KUKA KRL program: EPS_2_25716_MHDA01_A_20260123031854.src

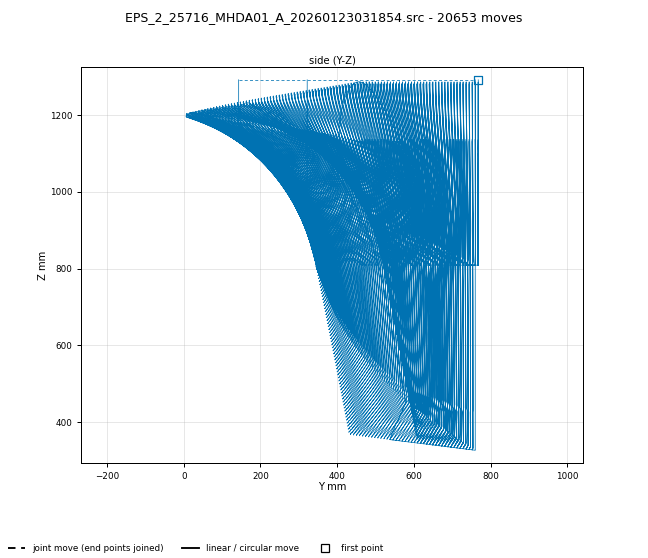
[picture p0: tool path of EPS_2_25716_MHDA01_A_20260123031854.src, 20653 of 20655 moves have a stored position in this frame; points joined in program order, loops and branches not executed]
&ACCESS RVP
&REL 4
&COMMENT QRS 19112012
&PARAM EDITMASK = *
DEF PART()
EXT BAS (BAS_COMMAND :IN,REAL :IN )
INT I
BAS (#INITMOV,0 )

;KUKA QRS Post kuka4.cps  Date:22-06-2017 !

File_ID=3001

QRS_PRE_INIT()

;Init var - Until changes are made in qrs_pre_init
Outlet_Square_prg=0
Inlet_1_Square_prg=0
Inlet_2_Square_prg=0
Inlet_3_Square_prg=0
Inlet_4_Square_prg=0
Inlet_5_Square_prg=0

Outlet_1={X 0.000, Y 457.000, Z 863.000, B 0.000, E1 0.000 }
Inlet_1={X 0.000, Y 457.000, Z 713.000, B 0.000, E1 245.000 }
Outlet_1_type=838
Inlet_1_type=838
;QRS#1=Sidecore dimensions
;QRS#2=825-33" Concrete
;QRS#3=825-33" Concrete
;QRS#4=
;QRS#5=
;QRS#6=
;QRS#7=
;QRS#8=
;QRS#9=S306-46
;QRS#10=S306-46
;QRS#11=
;QRS#12=
;QRS#13=
;QRS#14=
;QRS#15=
;QRS#16=1524x152x1753 5,75'
;QRS#17=EPS Height
;QRS#18=1282
;QRS#19=*
;QRS#20= UPDATED VERSION 22-06-2017
;QRS#21=*
Outlet_Square=0650
Inlet_1_Square=0650
Inlet_2_Square=0
Inlet_3_Square=0
Inlet_4_Square=0
Inlet_5_Square=0
Mill_Square=1
Outlet_Square_Prg=267
Inlet_1_Square_prg=267

QRS_INIT()

$ADVANCE=5

; T1
PTP {E1 173.029,E2 173.029}
PTP {X 0,Y 767.722,A -85,B 0,C 180,E1 173.029,E2 173.029,E3 0,E4 0,E5 0,E6 0}
QRS_SPEED_INIT()
LIN {X 0,Y 767.722,Z 1292,A -85,B 0,C 180,E1 173.029,E2 173.029,E3 0,E4 0,E5 0,E6 0} C_VEL
LIN {X 0,Y 767.722,Z 811.06,A -85,B 0,C 180,E1 173.029,E2 173.029} C_VEL
LIN {X 0,Y 767.749,Z 809.06,A -85,B 0,C 180,E1 173.179,E2 173.179} C_VEL
LIN {X 0,Y 767.812,Z 809.06,A -85,B 0,C 180,E1 173.458,E2 173.458} C_VEL
LIN {X 0,Y 767.844,Z 809.06,A -85,B 0,C 180,E1 177.201,E2 177.201} C_VEL
LIN {X 0,Y 767.885,Z 809.06,A -85,B 0,C 180,E1 180.933,E2 180.933} C_VEL
LIN {X 0,Y 767.853,Z 809.06,A -85,B 0,C 180,E1 184.668,E2 184.668} C_VEL
LIN {X 0,Y 767.842,Z 809.06,A -85,B 0,C 180,E1 188.423,E2 188.423} C_VEL
LIN {X 0,Y 767.815,Z 809.06,A -85,B 0,C 180,E1 192.216,E2 192.216} C_VEL
LIN {X 0,Y 767.835,Z 809.06,A -85,B 0,C 180,E1 196.207,E2 196.207} C_VEL
LIN {X 0,Y 767.767,Z 809.06,A -85,B 0,C 180,E1 199.988,E2 199.988} C_VEL
LIN {X 0,Y 767.76,Z 809.06,A -85,B 0,C 180,E1 204.012,E2 204.012} C_VEL
LIN {X 0,Y 767.747,Z 809.06,A -85,B 0,C 180,E1 208.167,E2 208.167} C_VEL
LIN {X 0,Y 767.299,Z 809.06,A -85,B 0,C 180,E1 210.325,E2 210.325} C_VEL
LIN {X 0,Y 767.722,Z 809.06,A -85,B 0,C 180,E1 212.492,E2 212.492} C_VEL
LIN {X 0,Y 767.413,Z 809.06,A -85,B 0,C 180,E1 213.849,E2 213.849} C_VEL
LIN {X 0,Y 767.746,Z 809.06,A -85,B 0,C 180,E1 217.099,E2 217.099} C_VEL
LIN {X 0,Y 767.186,Z 809.06,A -85,B 0,C 180,E1 220.04,E2 220.04} C_VEL
LIN {X 0,Y 767.672,Z 809.06,A -85,B 0,C 180,E1 221.87,E2 221.87} C_VEL
LIN {X 0,Y 767.699,Z 809.06,A -85,B 0,C 180,E1 222.901,E2 222.901} C_VEL
LIN {X 0,Y 767.698,Z 809.06,A -85,B 0,C 180,E1 224.426,E2 224.426} C_VEL
LIN {X 0,Y 767.66,Z 809.06,A -85,B 0,C 180,E1 225.572,E2 225.572} C_VEL
LIN {X 0,Y 767.698,Z 809.06,A -85,B 0,C 180,E1 229.916,E2 229.916} C_VEL
LIN {X 0,Y 767.769,Z 809.06,A -85,B 0,C 180,E1 230.595,E2 230.595} C_VEL
LIN {X 0,Y 767.848,Z 809.06,A -85,B 0,C 180,E1 233.269,E2 233.269} C_VEL
LIN {X 0,Y 766.331,Z 809.06,A -85,B 0,C 180,E1 233.48,E2 233.48} C_VEL
LIN {X 0,Y 767.104,Z 827.55,A -85,B 0,C 180,E1 233.745,E2 233.745} C_VEL
LIN {X 0,Y 767.17,Z 886.209,A -85,B 0,C 180,E1 234.412,E2 234.412} C_VEL
LIN {X 0,Y 767.458,Z 906.942,A -85,B 0,C 180,E1 234.685,E2 234.685} C_VEL
LIN {X 0,Y 767.407,Z 923.144,A -85,B 0,C 180,E1 234.938,E2 234.938} C_VEL
LIN {X 0,Y 767.212,Z 935.539,A -85,B 0,C 180,E1 235.164,E2 235.164} C_VEL
LIN {X 0,Y 767.339,Z 953.521,A -85,B 0,C 180,E1 235.567,E2 235.567} C_VEL
LIN {X 0,Y 767.292,Z 964.717,A -85,B 0,C 180,E1 235.849,E2 235.849} C_VEL
LIN {X 0,Y 767.46,Z 977.757,A -85,B 0,C 180,E1 236.229,E2 236.229} C_VEL
LIN {X 0,Y 767.482,Z 994.943,A -85,B 0,C 180,E1 236.765,E2 236.765} C_VEL
LIN {X 0,Y 767.407,Z 1008.2,A -85,B 0,C 180,E1 237.226,E2 237.226} C_VEL
LIN {X 0,Y 767.51,Z 1017.146,A -85,B 0,C 180,E1 237.568,E2 237.568} C_VEL
LIN {X 0,Y 767.581,Z 1032.615,A -85,B 0,C 180,E1 238.19,E2 238.19} C_VEL
LIN {X 0,Y 767.446,Z 1051.001,A -85,B 0,C 180,E1 239.004,E2 239.004} C_VEL
LIN {X 0,Y 767.587,Z 1068.192,A -85,B 0,C 180,E1 239.855,E2 239.855} C_VEL
LIN {X 0,Y 767.618,Z 1085.156,A -85,B 0,C 180,E1 240.771,E2 240.771} C_VEL
LIN {X 0,Y 767.607,Z 1101.948,A -85,B 0,C 180,E1 241.761,E2 241.761} C_VEL
LIN {X 0,Y 767.626,Z 1117.369,A -85,B 0,C 180,E1 242.75,E2 242.75} C_VEL
LIN {X 0,Y 767.651,Z 1132.728,A -85,B 0,C 180,E1 243.819,E2 243.819} C_VEL
LIN {X 0,Y 767.584,Z 1147.859,A -85,B 0,C 180,E1 244.959,E2 244.959} C_VEL
LIN {X 0,Y 767.612,Z 1160.458,A -85,B 0,C 180,E1 245.983,E2 245.983} C_VEL
LIN {X 0,Y 767.704,Z 1173.515,A -85,B 0,C 180,E1 247.13,E2 247.13} C_VEL
LIN {X 0,Y 767.583,Z 1186.75,A -85,B 0,C 180,E1 248.384,E2 248.384} C_VEL
LIN {X 0,Y 767.736,Z 1199.104,A -85,B 0,C 180,E1 249.665,E2 249.665} C_VEL
LIN {X 0,Y 767.55,Z 1210.953,A -85,B 0,C 180,E1 250.996,E2 250.996} C_VEL
LIN {X 0,Y 767.566,Z 1220.98,A -85,B 0,C 180,E1 252.225,E2 252.225} C_VEL
LIN {X 0,Y 767.803,Z 1230.047,A -85,B 0,C 180,E1 253.451,E2 253.451} C_VEL
LIN {X 0,Y 767.523,Z 1241.12,A -85,B 0,C 180,E1 255.092,E2 255.092} C_VEL
LIN {X 0,Y 767.763,Z 1249.724,A -85,B 0,C 180,E1 256.547,E2 256.547} C_VEL
LIN {X 0,Y 767.583,Z 1255.072,A -85,B 0,C 180,E1 257.542,E2 257.542} C_VEL
LIN {X 0,Y 767.466,Z 1258.642,A -85,B 0,C 180,E1 258.256,E2 258.256} C_VEL
LIN {X 0,Y 767.574,Z 1264.125,A -85,B 0,C 180,E1 259.446,E2 259.446} C_VEL
LIN {X 0,Y 767.772,Z 1266.941,A -85,B 0,C 180,E1 260.159,E2 260.159} C_VEL
LIN {X 0,Y 767.609,Z 1270.613,A -85,B 0,C 180,E1 261.103,E2 261.103} C_VEL
LIN {X 0,Y 767.526,Z 1275.33,A -85,B 0,C 180,E1 262.515,E2 262.515} C_VEL
LIN {X 0,Y 767.729,Z 1277.921,A -85,B 0,C 180,E1 263.457,E2 263.457} C_VEL
LIN {X 0,Y 767.753,Z 1279.763,A -85,B 0,C 180,E1 264.208,E2 264.208} C_VEL
LIN {X 0,Y 767.526,Z 1282.157,A -85,B 0,C 180,E1 265.33,E2 265.33} C_VEL
LIN {X 0,Y 767.596,Z 1283.961,A -85,B 0,C 180,E1 266.453,E2 266.453} C_VEL
LIN {X 0,Y 767.784,Z 1284.832,A -85,B 0,C 180,E1 267.201,E2 267.201} C_VEL
LIN {X 0,Y 767.485,Z 1286.213,A -85,B 0,C 180,E1 269.067,E2 269.067} C_VEL
LIN {X 0,Y 767.799,Z 1286.153,A -85,B 0,C 180,E1 270.932,E2 270.932} C_VEL
LIN {X 0,Y 767.787,Z 1284.832,A -85,B 0,C 180,E1 272.799,E2 272.799} C_VEL
LIN {X 0,Y 767.6,Z 1283.418,A -85,B 0,C 180,E1 273.921,E2 273.921} C_VEL
LIN {X 0,Y 767.502,Z 1282.163,A -85,B 0,C 180,E1 274.67,E2 274.67} C_VEL
LIN {X 0,Y 767.612,Z 1279.789,A -85,B 0,C 180,E1 275.793,E2 275.793} C_VEL
LIN {X 0,Y 767.819,Z 1277.906,A -85,B 0,C 180,E1 276.542,E2 276.542} C_VEL
LIN {X 0,Y 767.57,Z 1275.324,A -85,B 0,C 180,E1 277.484,E2 277.484} C_VEL
LIN {X 0,Y 767.464,Z 1270.637,A -85,B 0,C 180,E1 278.899,E2 278.899} C_VEL
LIN {X 0,Y 767.675,Z 1266.958,A -85,B 0,C 180,E1 279.842,E2 279.842} C_VEL
LIN {X 0,Y 767.812,Z 1264.091,A -85,B 0,C 180,E1 280.55,E2 280.55} C_VEL
LIN {X 0,Y 767.541,Z 1256.36,A -85,B 0,C 180,E1 282.22,E2 282.22} C_VEL
LIN {X 0,Y 767.797,Z 1247.861,A -85,B 0,C 180,E1 283.778,E2 283.778} C_VEL
LIN {X 0,Y 767.526,Z 1239.921,A -85,B 0,C 180,E1 285.1,E2 285.1} C_VEL
LIN {X 0,Y 767.65,Z 1230.061,A -85,B 0,C 180,E1 286.552,E2 286.552} C_VEL
LIN {X 0,Y 767.763,Z 1224.604,A -85,B 0,C 180,E1 287.281,E2 287.281} C_VEL
LIN {X 0,Y 767.618,Z 1219.008,A -85,B 0,C 180,E1 288.018,E2 288.018} C_VEL
LIN {X 0,Y 767.578,Z 1208.865,A -85,B 0,C 180,E1 289.25,E2 289.25} C_VEL
LIN {X 0,Y 767.782,Z 1196.924,A -85,B 0,C 180,E1 290.566,E2 290.566} C_VEL
LIN {X 0,Y 767.586,Z 1184.113,A -85,B 0,C 180,E1 291.872,E2 291.872} C_VEL
LIN {X 0,Y 767.66,Z 1172.11,A -85,B 0,C 180,E1 292.998,E2 292.998} C_VEL
LIN {X 0,Y 767.691,Z 1158.934,A -85,B 0,C 180,E1 294.142,E2 294.142} C_VEL
LIN {X 0,Y 767.62,Z 1144.01,A -85,B 0,C 180,E1 295.338,E2 295.338} C_VEL
LIN {X 0,Y 767.652,Z 1129.639,A -85,B 0,C 180,E1 296.401,E2 296.401} C_VEL
LIN {X 0,Y 767.615,Z 1114.367,A -85,B 0,C 180,E1 297.447,E2 297.447} C_VEL
LIN {X 0,Y 767.599,Z 1098.637,A -85,B 0,C 180,E1 298.44,E2 298.44} C_VEL
LIN {X 0,Y 767.566,Z 1083.423,A -85,B 0,C 180,E1 299.33,E2 299.33} C_VEL
LIN {X 0,Y 767.575,Z 1064.92,A -85,B 0,C 180,E1 300.312,E2 300.312} C_VEL
LIN {X 0,Y 767.441,Z 1046.6,A -85,B 0,C 180,E1 301.2,E2 301.2} C_VEL
LIN {X 0,Y 767.574,Z 1029.388,A -85,B 0,C 180,E1 301.947,E2 301.947} C_VEL
LIN {X 0,Y 767.522,Z 1009.76,A -85,B 0,C 180,E1 302.714,E2 302.714} C_VEL
LIN {X 0,Y 767.358,Z 997.436,A -85,B 0,C 180,E1 303.153,E2 303.153} C_VEL
LIN {X 0,Y 767.471,Z 988.18,A -85,B 0,C 180,E1 303.452,E2 303.452} C_VEL
LIN {X 0,Y 767.491,Z 969.899,A -85,B 0,C 180,E1 303.999,E2 303.999} C_VEL
LIN {X 0,Y 767.246,Z 953.494,A -85,B 0,C 180,E1 304.438,E2 304.438} C_VEL
LIN {X 0,Y 767.411,Z 935.529,A -85,B 0,C 180,E1 304.826,E2 304.826} C_VEL
LIN {X 0,Y 767.255,Z 918.227,A -85,B 0,C 180,E1 305.152,E2 305.152} C_VEL
LIN {X 0,Y 767.195,Z 912.098,A -85,B 0,C 180,E1 305.255,E2 305.255} C_VEL
LIN {X 0,Y 767.34,Z 895.861,A -85,B 0,C 180,E1 305.467,E2 305.467} C_VEL
LIN {X 0,Y 767.184,Z 847.286,A -85,B 0,C 180,E1 306.027,E2 306.027} C_VEL
LIN {X 0,Y 766.354,Z 809.06,A -85,B 0,C 180,E1 306.518,E2 306.518} C_VEL
LIN {X 0,Y 767.867,Z 809.06,A -85,B 0,C 180,E1 307.025,E2 307.025} C_VEL
LIN {X 0,Y 767.157,Z 809.06,A -85,B 0,C 180,E1 310.036,E2 310.036} C_VEL
LIN {X 0,Y 767.638,Z 809.06,A -85,B 0,C 180,E1 311.871,E2 311.871} C_VEL
LIN {X 0,Y 767.679,Z 809.06,A -85,B 0,C 180,E1 312.899,E2 312.899} C_VEL
LIN {X 0,Y 767.687,Z 809.06,A -85,B 0,C 180,E1 314.425,E2 314.425} C_VEL
LIN {X 0,Y 767.662,Z 809.06,A -85,B 0,C 180,E1 315.572,E2 315.572} C_VEL
LIN {X 0,Y 767.695,Z 809.06,A -85,B 0,C 180,E1 319.914,E2 319.914} C_VEL
LIN {X 0,Y 767.699,Z 809.06,A -85,B 0,C 180,E1 320.59,E2 320.59} C_VEL
LIN {X 0,Y 767.222,Z 809.06,A -85,B 0,C 180,E1 322.952,E2 322.952} C_VEL
LIN {X 0,Y 767.706,Z 809.06,A -85,B 0,C 180,E1 325.267,E2 325.267} C_VEL
LIN {X 0,Y 767.75,Z 809.06,A -85,B 0,C 180,E1 329.62,E2 329.62} C_VEL
LIN {X 0,Y 767.63,Z 809.06,A -85,B 0,C 180,E1 333.924,E2 333.924} C_VEL
LIN {X 0,Y 767.153,Z 809.06,A -85,B 0,C 180,E1 335.967,E2 335.967} C_VEL
LIN {X 0,Y 767.108,Z 809.06,A -85,B 0,C 180,E1 338.214,E2 338.214} C_VEL
LIN {X 0,Y 767.721,Z 809.06,A -85,B 0,C 180,E1 340.011,E2 340.011} C_VEL
LIN {X 0,Y 767.197,Z 809.06,A -85,B 0,C 180,E1 343.956,E2 343.956} C_VEL
LIN {X 0,Y 767.618,Z 809.06,A -85,B 0,C 180,E1 345.865,E2 345.865} C_VEL
LIN {X 0,Y 767.838,Z 809.06,A -85,B 0,C 180,E1 350.26,E2 350.26} C_VEL
LIN {X 0,Y 767.551,Z 809.06,A -85,B 0,C 180,E1 350.49,E2 350.49} C_VEL
LIN {X 0,Y 766.698,Z 809.096,A -85,B 0,C 180,E1 350.63,E2 350.63} C_VEL
LIN {X 0,Y 767.228,Z 811.332,A -85,B 0,C 180,E1 350.713,E2 350.713} C_VEL
LIN {X 0,Y 767.311,Z 825.627,A -85,B 0,C 180,E1 351.111,E2 351.111} C_VEL
LIN {X 0,Y 767.555,Z 844.038,A -85,B 0,C 180,E1 351.692,E2 351.692} C_VEL
LIN {X 0,Y 767.554,Z 863.959,A -85,B 0,C 180,E1 352.398,E2 352.398} C_VEL
LIN {X 0,Y 767.461,Z 878.632,A -85,B 0,C 180,E1 352.973,E2 352.973} C_VEL
LIN {X 0,Y 767.581,Z 900.185,A -85,B 0,C 180,E1 353.925,E2 353.925} C_VEL
LIN {X 0,Y 767.495,Z 917.486,A -85,B 0,C 180,E1 354.768,E2 354.768} C_VEL
LIN {X 0,Y 767.597,Z 934.813,A -85,B 0,C 180,E1 355.705,E2 355.705} C_VEL
LIN {X 0,Y 767.629,Z 952.205,A -85,B 0,C 180,E1 356.733,E2 356.733} C_VEL
LIN {X 0,Y 767.617,Z 968.181,A -85,B 0,C 180,E1 357.761,E2 357.761} C_VEL
LIN {X 0,Y 767.615,Z 982.927,A -85,B 0,C 180,E1 358.787,E2 358.787} C_VEL
LIN {X 0,Y 767.661,Z 997.734,A -85,B 0,C 180,E1 359.907,E2 359.907} C_VEL
LIN {X 0,Y 767.561,Z 1011.487,A -85,B 0,C 180,E1 361.026,E2 361.026} C_VEL
LIN {X 0,Y 767.601,Z 1023.209,A -85,B 0,C 180,E1 362.053,E2 362.053} C_VEL
LIN {X 0,Y 767.724,Z 1036.904,A -85,B 0,C 180,E1 363.36,E2 363.36} C_VEL
LIN {X 0,Y 767.584,Z 1049.581,A -85,B 0,C 180,E1 364.669,E2 364.669} C_VEL
LIN {X 0,Y 767.729,Z 1059.606,A -85,B 0,C 180,E1 365.792,E2 365.792} C_VEL
LIN {X 0,Y 767.674,Z 1065.767,A -85,B 0,C 180,E1 366.543,E2 366.543} C_VEL
LIN {X 0,Y 767.525,Z 1072.035,A -85,B 0,C 180,E1 367.321,E2 367.321} C_VEL
LIN {X 0,Y 767.563,Z 1081.893,A -85,B 0,C 180,E1 368.662,E2 368.662} C_VEL
LIN {X 0,Y 767.797,Z 1089.765,A -85,B 0,C 180,E1 369.84,E2 369.84} C_VEL
LIN {X 0,Y 767.53,Z 1099.791,A -85,B 0,C 180,E1 371.505,E2 371.505} C_VEL
LIN {X 0,Y 767.778,Z 1107.286,A -85,B 0,C 180,E1 372.933,E2 372.933} C_VEL
LIN {X 0,Y 767.522,Z 1112.962,A -85,B 0,C 180,E1 374.137,E2 374.137} C_VEL
LIN {X 0,Y 767.554,Z 1119.271,A -85,B 0,C 180,E1 375.681,E2 375.681} C_VEL
LIN {X 0,Y 767.779,Z 1122.233,A -85,B 0,C 180,E1 376.55,E2 376.55} C_VEL
LIN {X 0,Y 767.605,Z 1125.485,A -85,B 0,C 180,E1 377.529,E2 377.529} C_VEL
LIN {X 0,Y 767.52,Z 1128.22,A -85,B 0,C 180,E1 378.512,E2 378.512} C_VEL
LIN {X 0,Y 767.661,Z 1130.538,A -85,B 0,C 180,E1 379.495,E2 379.495} C_VEL
LIN {X 0,Y 767.803,Z 1131.516,A -85,B 0,C 180,E1 379.987,E2 379.987} C_VEL
LIN {X 0,Y 767.622,Z 1133.359,A -85,B 0,C 180,E1 381.002,E2 381.002} C_VEL
LIN {X 0,Y 767.515,Z 1134.743,A -85,B 0,C 180,E1 381.993,E2 381.993} C_VEL
LIN {X 0,Y 767.742,Z 1136.161,A -85,B 0,C 180,E1 384.013,E2 384.013} C_VEL
LIN {X 0,Y 767.561,Z 1136.046,A -85,B 0,C 180,E1 386.432,E2 386.432} C_VEL
LIN {X 0,Y 767.728,Z 1135.41,A -85,B 0,C 180,E1 387.115,E2 387.115} C_VEL
LIN {X 0,Y 767.578,Z 1134.408,A -85,B 0,C 180,E1 388.174,E2 388.174} C_VEL
LIN {X 0,Y 767.503,Z 1132.862,A -85,B 0,C 180,E1 389.222,E2 389.222} C_VEL
LIN {X 0,Y 767.703,Z 1130.624,A -85,B 0,C 180,E1 390.374,E2 390.374} C_VEL
LIN {X 0,Y 767.841,Z 1129.529,A -85,B 0,C 180,E1 390.843,E2 390.843} C_VEL
LIN {X 0,Y 767.562,Z 1126.749,A -85,B 0,C 180,E1 391.948,E2 391.948} C_VEL
LIN {X 0,Y 767.533,Z 1123.994,A -85,B 0,C 180,E1 392.855,E2 392.855} C_VEL
LIN {X 0,Y 767.718,Z 1120.411,A -85,B 0,C 180,E1 393.906,E2 393.906} C_VEL
LIN {X 0,Y 767.83,Z 1118.878,A -85,B 0,C 180,E1 394.312,E2 394.312} C_VEL
LIN {X 0,Y 767.525,Z 1113.89,A -85,B 0,C 180,E1 395.57,E2 395.57} C_VEL
LIN {X 0,Y 767.613,Z 1106.806,A -85,B 0,C 180,E1 397.087,E2 397.087} C_VEL
LIN {X 0,Y 767.833,Z 1102.272,A -85,B 0,C 180,E1 397.927,E2 397.927} C_VEL
LIN {X 0,Y 767.662,Z 1099.064,A -85,B 0,C 180,E1 398.536,E2 398.536} C_VEL
LIN {X 0,Y 767.546,Z 1089.659,A -85,B 0,C 180,E1 400.093,E2 400.093} C_VEL
LIN {X 0,Y 767.784,Z 1080.734,A -85,B 0,C 180,E1 401.412,E2 401.412} C_VEL
LIN {X 0,Y 767.553,Z 1069.535,A -85,B 0,C 180,E1 402.911,E2 402.911} C_VEL
LIN {X 0,Y 767.733,Z 1058.591,A -85,B 0,C 180,E1 404.231,E2 404.231} C_VEL
LIN {X 0,Y 767.681,Z 1050.536,A -85,B 0,C 180,E1 405.131,E2 405.131} C_VEL
LIN {X 0,Y 767.59,Z 1044.661,A -85,B 0,C 180,E1 405.758,E2 405.758} C_VEL
LIN {X 0,Y 767.609,Z 1035.423,A -85,B 0,C 180,E1 406.703,E2 406.703} C_VEL
LIN {X 0,Y 767.737,Z 1022.981,A -85,B 0,C 180,E1 407.874,E2 407.874} C_VEL
LIN {X 0,Y 767.592,Z 1008.626,A -85,B 0,C 180,E1 409.125,E2 409.125} C_VEL
LIN {X 0,Y 767.659,Z 994.663,A -85,B 0,C 180,E1 410.243,E2 410.243} C_VEL
LIN {X 0,Y 767.618,Z 979.599,A -85,B 0,C 180,E1 411.36,E2 411.36} C_VEL
LIN {X 0,Y 767.591,Z 964.172,A -85,B 0,C 180,E1 412.415,E2 412.415} C_VEL
LIN {X 0,Y 767.548,Z 949.165,A -85,B 0,C 180,E1 413.367,E2 413.367} C_VEL
LIN {X 0,Y 767.605,Z 932.06,A -85,B 0,C 180,E1 414.356,E2 414.356} C_VEL
LIN {X 0,Y 767.575,Z 915.036,A -85,B 0,C 180,E1 415.262,E2 415.262} C_VEL
LIN {X 0,Y 767.548,Z 900.158,A -85,B 0,C 180,E1 415.988,E2 415.988} C_VEL
LIN {X 0,Y 767.557,Z 879.517,A -85,B 0,C 180,E1 416.897,E2 416.897} C_VEL
LIN {X 0,Y 767.355,Z 861.124,A -85,B 0,C 180,E1 417.63,E2 417.63} C_VEL
LIN {X 0,Y 767.531,Z 840.76,A -85,B 0,C 180,E1 418.326,E2 418.326} C_VEL
LIN {X 0,Y 767.41,Z 820.126,A -85,B 0,C 180,E1 418.952,E2 418.952} C_VEL
LIN {X 0,Y 767.15,Z 809.2,A -85,B 0,C 180,E1 419.255,E2 419.255} C_VEL
LIN {X 0,Y 767.208,Z 809.06,A -85,B 0,C 180,E1 419.266,E2 419.266} C_VEL
LIN {X 0,Y 767.722,Z 809.06,A -85,B 0,C 180,E1 419.356,E2 419.356} C_VEL
LIN {X 0,Y 767.842,Z 809.06,A -85,B 0,C 180,E1 419.513,E2 419.513} C_VEL
LIN {X 0,Y 767.638,Z 809.06,A -85,B 0,C 180,E1 423.925,E2 423.925} C_VEL
LIN {X 0,Y 767.153,Z 809.06,A -85,B 0,C 180,E1 425.968,E2 425.968} C_VEL
LIN {X 0,Y 767.097,Z 809.06,A -85,B 0,C 180,E1 428.219,E2 428.219} C_VEL
LIN {X 0,Y 767.703,Z 809.06,A -85,B 0,C 180,E1 430.011,E2 430.011} C_VEL
LIN {X 0,Y 767.177,Z 809.06,A -85,B 0,C 180,E1 433.965,E2 433.965} C_VEL
LIN {X 0,Y 767.655,Z 809.06,A -85,B 0,C 180,E1 435.866,E2 435.866} C_VEL
LIN {X 0,Y 767.851,Z 809.06,A -85,B 0,C 180,E1 439.687,E2 439.687} C_VEL
LIN {X 0,Y 767.825,Z 809.06,A -85,B 0,C 180,E1 443.458,E2 443.458} C_VEL
LIN {X 0,Y 767.805,Z 809.06,A -85,B 0,C 180,E1 447.201,E2 447.201} C_VEL
LIN {X 0,Y 767.788,Z 809.06,A -85,B 0,C 180,E1 450.933,E2 450.933} C_VEL
LIN {X 0,Y 767.798,Z 809.06,A -85,B 0,C 180,E1 454.668,E2 454.668} C_VEL
LIN {X 0,Y 767.818,Z 809.06,A -85,B 0,C 180,E1 458.423,E2 458.423} C_VEL
LIN {X 0,Y 767.83,Z 809.06,A -85,B 0,C 180,E1 462.215,E2 462.215} C_VEL
LIN {X 0,Y 767.855,Z 809.06,A -85,B 0,C 180,E1 466.21,E2 466.21} C_VEL
LIN {X 0,Y 767.775,Z 809.06,A -85,B 0,C 180,E1 469.988,E2 469.988} C_VEL
LIN {X 0,Y 767.749,Z 809.06,A -85,B 0,C 180,E1 474.013,E2 474.013} C_VEL
LIN {X 0,Y 767.745,Z 809.06,A -85,B 0,C 180,E1 478.167,E2 478.167} C_VEL
LIN {X 0,Y 767.323,Z 809.06,A -85,B 0,C 180,E1 480.323,E2 480.323} C_VEL
LIN {X 0,Y 767.748,Z 809.06,A -85,B 0,C 180,E1 482.49,E2 482.49} C_VEL
LIN {X 0,Y 767.436,Z 809.06,A -85,B 0,C 180,E1 483.851,E2 483.851} C_VEL
LIN {X 0,Y 767.74,Z 809.06,A -85,B 0,C 180,E1 487.098,E2 487.098} C_VEL
LIN {X 0,Y 767.15,Z 809.06,A -85,B 0,C 180,E1 490.036,E2 490.036} C_VEL
LIN {X 0,Y 767.63,Z 809.06,A -85,B 0,C 180,E1 491.873,E2 491.873} C_VEL
LIN {X 0,Y 767.654,Z 809.06,A -85,B 0,C 180,E1 492.897,E2 492.897} C_VEL
LIN {X 0,Y 767.673,Z 809.06,A -85,B 0,C 180,E1 494.427,E2 494.427} C_VEL
LIN {X 0,Y 767.645,Z 809.06,A -85,B 0,C 180,E1 495.571,E2 495.571} C_VEL
LIN {X 0,Y 767.658,Z 809.06,A -85,B 0,C 180,E1 499.918,E2 499.918} C_VEL
LIN {X 0,Y 767.644,Z 809.06,A -85,B 0,C 180,E1 500.587,E2 500.587} C_VEL
LIN {X 0,Y 767.207,Z 809.06,A -85,B 0,C 180,E1 502.954,E2 502.954} C_VEL
LIN {X 0,Y 767.702,Z 809.06,A -85,B 0,C 180,E1 505.267,E2 505.267} C_VEL
LIN {X 0,Y 767.777,Z 809.06,A -85,B 0,C 180,E1 509.618,E2 509.618} C_VEL
LIN {X 0,Y 767.797,Z 809.06,A -85,B 0,C 180,E1 513.534,E2 513.534} C_VEL
LIN {X 0,Y 767.795,Z 809.06,A -85,B 0,C 180,E1 513.93,E2 513.93} C_VEL
LIN {X 0,Y 767.807,Z 809.06,A -85,B 0,C 180,E1 518.016,E2 518.016} C_VEL
LIN {X 0,Y 767.828,Z 809.06,A -85,B 0,C 180,E1 521.986,E2 521.986} C_VEL
LIN {X 0,Y 767.5,Z 809.06,A -85,B 0,C 180,E1 523.93,E2 523.93} C_VEL
LIN {X 0,Y 767.62,Z 809.06,A -85,B 0,C 180,E1 525.865,E2 525.865} C_VEL
LIN {X 0,Y 767.81,Z 809.06,A -85,B 0,C 180,E1 529.686,E2 529.686} C_VEL
LIN {X 0,Y 767.749,Z 809.06,A -85,B 0,C 180,E1 533.179,E2 533.179} C_VEL
LIN {X 0,Y 765.187,Z 809.06,A -85,B 0,C 180,E1 534.137,E2 534.137} C_VEL
LIN {X 0,Y 759.627,Z 809.06,A -85,B 0,C 180,E1 535.565,E2 535.565} C_VEL
LIN {X 0,Y 759.547,Z 809.06,A -85,B 0,C 180,E1 535.73,E2 535.73} C_VEL
LIN {X 0,Y 759.695,Z 809.06,A -85,B 0,C 180,E1 540,E2 540} C_VEL
LIN {X 0,Y 759.906,Z 809.06,A -85,B 0,C 180,E1 544.562,E2 544.562} C_VEL
LIN {X 0,Y 759.673,Z 809.06,A -85,B 0,C 180,E1 549.156,E2 549.156} C_VEL
LIN {X 0,Y 759.479,Z 809.06,A -85,B 0,C 180,E1 553.813,E2 553.813} C_VEL
LIN {X 0,Y 759.572,Z 809.06,A -85,B 0,C 180,E1 557.361,E2 557.361} C_VEL
LIN {X 0,Y 759.541,Z 809.06,A -85,B 0,C 180,E1 560.983,E2 560.983} C_VEL
LIN {X 0,Y 759.596,Z 809.06,A -85,B 0,C 180,E1 564.692,E2 564.692} C_VEL
LIN {X 0,Y 759.591,Z 809.06,A -85,B 0,C 180,E1 568.912,E2 568.912} C_VEL
LIN {X 0,Y 759.592,Z 809.06,A -85,B 0,C 180,E1 573.324,E2 573.324} C_VEL
LIN {X 0,Y 759.452,Z 809.06,A -85,B 0,C 180,E1 578.081,E2 578.081} C_VEL
LIN {X 0,Y 759.796,Z 809.06,A -85,B 0,C 180,E1 582.615,E2 582.615} C_VEL
LIN {X 0,Y 759.626,Z 809.06,A -85,B 0,C 180,E1 585.869,E2 585.869} C_VEL
LIN {X 0,Y 759.822,Z 809.06,A -85,B 0,C 180,E1 590.856,E2 590.856} C_VEL
LIN {X 0,Y 759.872,Z 809.447,A -85,B 0,C 180,E1 593.134,E2 593.134} C_VEL
LIN {X 0,Y 760.755,Z 883.004,A -85,B 0,C 180,E1 594.029,E2 594.029} C_VEL
LIN {X 0,Y 760.679,Z 936.538,A -85,B 0,C 180,E1 594.842,E2 594.842} C_VEL
LIN {X 0,Y 760.763,Z 980.986,A -85,B 0,C 180,E1 595.991,E2 595.991} C_VEL
LIN {X 0,Y 760.667,Z 1026.204,A -85,B 0,C 180,E1 597.601,E2 597.601} C_VEL
LIN {X 0,Y 760.489,Z 1068.344,A -85,B 0,C 180,E1 599.552,E2 599.552} C_VEL
LIN {X 0,Y 760.286,Z 1112.591,A -85,B 0,C 180,E1 602.151,E2 602.151} C_VEL
LIN {X 0,Y 760.061,Z 1149.729,A -85,B 0,C 180,E1 604.848,E2 604.848} C_VEL
LIN {X 0,Y 759.948,Z 1184.696,A -85,B 0,C 180,E1 607.952,E2 607.952} C_VEL
LIN {X 0,Y 759.78,Z 1213.754,A -85,B 0,C 180,E1 611.14,E2 611.14} C_VEL
LIN {X 0,Y 759.76,Z 1237.856,A -85,B 0,C 180,E1 614.42,E2 614.42} C_VEL
LIN {X 0,Y 759.717,Z 1256.533,A -85,B 0,C 180,E1 617.649,E2 617.649} C_VEL
LIN {X 0,Y 759.799,Z 1270.399,A -85,B 0,C 180,E1 620.841,E2 620.841} C_VEL
LIN {X 0,Y 759.847,Z 1280.559,A -85,B 0,C 180,E1 624.289,E2 624.289} C_VEL
LIN {X 0,Y 759.757,Z 1285.87,A -85,B 0,C 180,E1 627.716,E2 627.716} C_VEL
LIN {X 0,Y 759.887,Z 1286.67,A -85,B 0,C 180,E1 631.135,E2 631.135} C_VEL
LIN {X 0,Y 759.654,Z 1282.919,A -85,B 0,C 180,E1 634.559,E2 634.559} C_VEL
LIN {X 0,Y 759.613,Z 1274.303,A -85,B 0,C 180,E1 638,E2 638} C_VEL
LIN {X 0,Y 759.74,Z 1260.714,A -85,B 0,C 180,E1 641.467,E2 641.467} C_VEL
LIN {X 0,Y 759.748,Z 1243.488,A -85,B 0,C 180,E1 644.685,E2 644.685} C_VEL
LIN {X 0,Y 759.835,Z 1219.927,A -85,B 0,C 180,E1 648.098,E2 648.098} C_VEL
LIN {X 0,Y 759.935,Z 1189.309,A -85,B 0,C 180,E1 651.578,E2 651.578} C_VEL
LIN {X 0,Y 760.098,Z 1155.61,A -85,B 0,C 180,E1 654.67,E2 654.67} C_VEL
LIN {X 0,Y 760.271,Z 1116.487,A -85,B 0,C 180,E1 657.597,E2 657.597} C_VEL
LIN {X 0,Y 760.442,Z 1073.092,A -85,B 0,C 180,E1 660.192,E2 660.192} C_VEL
LIN {X 0,Y 760.676,Z 1030.037,A -85,B 0,C 180,E1 662.245,E2 662.245} C_VEL
LIN {X 0,Y 760.773,Z 984.117,A -85,B 0,C 180,E1 663.912,E2 663.912} C_VEL
LIN {X 0,Y 760.849,Z 940.168,A -85,B 0,C 180,E1 665.073,E2 665.073} C_VEL
LIN {X 0,Y 760.917,Z 896.088,A -85,B 0,C 180,E1 665.809,E2 665.809} C_VEL
LIN {X 0,Y 759.649,Z 811.384,A -85,B 0,C 180,E1 666.856,E2 666.856} C_VEL
LIN {X 0,Y 759.59,Z 809.06,A -85,B 0,C 180,E1 666.966,E2 666.966} C_VEL
LIN {X 0,Y 759.744,Z 809.06,A -85,B 0,C 180,E1 672.619,E2 672.619} C_VEL
LIN {X 0,Y 759.629,Z 809.06,A -85,B 0,C 180,E1 675.877,E2 675.877} C_VEL
LIN {X 0,Y 759.693,Z 809.06,A -85,B 0,C 180,E1 680.863,E2 680.863} C_VEL
LIN {X 0,Y 759.463,Z 809.06,A -85,B 0,C 180,E1 686.146,E2 686.146} C_VEL
LIN {X 0,Y 759.608,Z 809.06,A -85,B 0,C 180,E1 690.178,E2 690.178} C_VEL
LIN {X 0,Y 759.671,Z 809.06,A -85,B 0,C 180,E1 694.05,E2 694.05} C_VEL
LIN {X 0,Y 759.69,Z 809.06,A -85,B 0,C 180,E1 700.237,E2 700.237} C_VEL
LIN {X 0,Y 759.581,Z 809.06,A -85,B 0,C 180,E1 706.189,E2 706.189} C_VEL
LIN {X 0,Y 759.914,Z 809.06,A -85,B 0,C 180,E1 710.269,E2 710.269} C_VEL
LIN {X 0,Y 760.78,Z 860.413,A -85,B 0,C 180,E1 711.936,E2 711.936} C_VEL
LIN {X 0,Y 760.521,Z 904.257,A -85,B 0,C 180,E1 713.806,E2 713.806} C_VEL
LIN {X 0,Y 760.366,Z 948.753,A -85,B 0,C 180,E1 716.225,E2 716.225} C_VEL
LIN {X 0,Y 760.157,Z 987.541,A -85,B 0,C 180,E1 718.861,E2 718.861} C_VEL
LIN {X 0,Y 759.98,Z 1023.646,A -85,B 0,C 180,E1 721.851,E2 721.851} C_VEL
LIN {X 0,Y 759.894,Z 1055.586,A -85,B 0,C 180,E1 725.133,E2 725.133} C_VEL
LIN {X 0,Y 759.722,Z 1080.587,A -85,B 0,C 180,E1 728.29,E2 728.29} C_VEL
LIN {X 0,Y 759.678,Z 1100.531,A -85,B 0,C 180,E1 731.472,E2 731.472} C_VEL
LIN {X 0,Y 759.629,Z 1116.016,A -85,B 0,C 180,E1 734.691,E2 734.691} C_VEL
LIN {X 0,Y 759.691,Z 1127.341,A -85,B 0,C 180,E1 737.956,E2 737.956} C_VEL
LIN {X 0,Y 759.759,Z 1133.875,A -85,B 0,C 180,E1 740.976,E2 740.976} C_VEL
LIN {X 0,Y 759.711,Z 1136.928,A -85,B 0,C 180,E1 744.687,E2 744.687} C_VEL
LIN {X 0,Y 759.843,Z 1135.891,A -85,B 0,C 180,E1 747.217,E2 747.217} C_VEL
LIN {X 0,Y 759.847,Z 1131.006,A -85,B 0,C 180,E1 750.469,E2 750.469} C_VEL
LIN {X 0,Y 759.92,Z 1120.179,A -85,B 0,C 180,E1 754.174,E2 754.174} C_VEL
LIN {X 0,Y 759.967,Z 1102.56,A -85,B 0,C 180,E1 758.05,E2 758.05} C_VEL
LIN {X 0,Y 759.953,Z 1080.89,A -85,B 0,C 180,E1 761.573,E2 761.573} C_VEL
LIN {X 0,Y 759.959,Z 1053.181,A -85,B 0,C 180,E1 765.047,E2 765.047} C_VEL
LIN {X 0,Y 760.072,Z 1021.52,A -85,B 0,C 180,E1 768.248,E2 768.248} C_VEL
LIN {X 0,Y 760.212,Z 982.575,A -85,B 0,C 180,E1 771.424,E2 771.424} C_VEL
LIN {X 0,Y 760.337,Z 942.383,A -85,B 0,C 180,E1 774.062,E2 774.062} C_VEL
LIN {X 0,Y 760.57,Z 898.635,A -85,B 0,C 180,E1 776.378,E2 776.378} C_VEL
LIN {X 0,Y 760.677,Z 852.483,A -85,B 0,C 180,E1 778.26,E2 778.26} C_VEL
LIN {X 0,Y 759.908,Z 809.515,A -85,B 0,C 180,E1 779.62,E2 779.62} C_VEL
LIN {X 0,Y 759.678,Z 809.06,A -85,B 0,C 180,E1 784.055,E2 784.055} C_VEL
LIN {X 0,Y 759.67,Z 809.06,A -85,B 0,C 180,E1 790.241,E2 790.241} C_VEL
LIN {X 0,Y 759.635,Z 809.06,A -85,B 0,C 180,E1 796.195,E2 796.195} C_VEL
LIN {X 0,Y 759.96,Z 809.06,A -85,B 0,C 180,E1 799.696,E2 799.696} C_VEL
LIN {X 0,Y 759.635,Z 809.06,A -85,B 0,C 180,E1 804.297,E2 804.297} C_VEL
LIN {X 0,Y 759.5,Z 809.06,A -85,B 0,C 180,E1 808.865,E2 808.865} C_VEL
LIN {X 0,Y 759.528,Z 809.06,A -85,B 0,C 180,E1 812.285,E2 812.285} C_VEL
LIN {X 0,Y 759.539,Z 809.06,A -85,B 0,C 180,E1 815.92,E2 815.92} C_VEL
LIN {X 0,Y 759.529,Z 809.06,A -85,B 0,C 180,E1 820.319,E2 820.319} C_VEL
LIN {X 0,Y 759.505,Z 809.06,A -85,B 0,C 180,E1 823.817,E2 823.817} C_VEL
LIN {X 0,Y 759.601,Z 809.06,A -85,B 0,C 180,E1 827.366,E2 827.366} C_VEL
LIN {X 0,Y 759.536,Z 809.06,A -85,B 0,C 180,E1 830.988,E2 830.988} C_VEL
LIN {X 0,Y 759.581,Z 809.06,A -85,B 0,C 180,E1 834.698,E2 834.698} C_VEL
LIN {X 0,Y 759.451,Z 809.06,A -85,B 0,C 180,E1 839.834,E2 839.834} C_VEL
LIN {X 0,Y 759.534,Z 809.06,A -85,B 0,C 180,E1 843.857,E2 843.857} C_VEL
LIN {X 0,Y 759.437,Z 809.06,A -85,B 0,C 180,E1 848.089,E2 848.089} C_VEL
LIN {X 0,Y 759.754,Z 809.06,A -85,B 0,C 180,E1 852.621,E2 852.621} C_VEL
LIN {X 0,Y 759.605,Z 809.06,A -85,B 0,C 180,E1 855.877,E2 855.877} C_VEL
LIN {X 0,Y 759.646,Z 809.06,A -85,B 0,C 180,E1 860.882,E2 860.882} C_VEL
LIN {X 0,Y 759.479,Z 809.06,A -85,B 0,C 180,E1 866.148,E2 866.148} C_VEL
LIN {X 0,Y 759.484,Z 809.06,A -85,B 0,C 180,E1 871.103,E2 871.103} C_VEL
LIN {X 0,Y 759.854,Z 809.06,A -85,B 0,C 180,E1 874.058,E2 874.058} C_VEL
LIN {X 0,Y 759.583,Z 809.06,A -85,B 0,C 180,E1 879.019,E2 879.019} C_VEL
LIN {X 0,Y 759.609,Z 809.06,A -85,B 0,C 180,E1 883.831,E2 883.831} C_VEL
LIN {X 0,Y 759.517,Z 809.06,A -85,B 0,C 180,E1 888.525,E2 888.525} C_VEL
LIN {X 0,Y 759.573,Z 809.06,A -85,B 0,C 180,E1 891.996,E2 891.996} C_VEL
LIN {X 0,Y 759.547,Z 809.06,A -85,B 0,C 180,E1 895.73,E2 895.73} C_VEL
LIN {X 0,Y 758.374,Z 809.06,A -85,B 0,C 180,E1 896.383,E2 896.383} C_VEL
LIN {X 0,Y 751.831,Z 809.06,A -85,B 0,C 180,E1 898.153,E2 898.153} C_VEL
LIN {X 0,Y 751.716,Z 809.06,A -85,B 0,C 180,E1 898.321,E2 898.321} C_VEL
LIN {X 0,Y 751.718,Z 809.06,A -85,B 0,C 180,E1 902.304,E2 902.304} C_VEL
LIN {X 0,Y 751.741,Z 809.06,A -85,B 0,C 180,E1 905.768,E2 905.768} C_VEL
LIN {X 0,Y 751.641,Z 809.06,A -85,B 0,C 180,E1 909.889,E2 909.889} C_VEL
LIN {X 0,Y 751.573,Z 809.06,A -85,B 0,C 180,E1 913.961,E2 913.961} C_VEL
LIN {X 0,Y 751.642,Z 809.06,A -85,B 0,C 180,E1 917.55,E2 917.55} C_VEL
LIN {X 0,Y 751.589,Z 809.06,A -85,B 0,C 180,E1 921.216,E2 921.216} C_VEL
LIN {X 0,Y 751.578,Z 809.06,A -85,B 0,C 180,E1 925.203,E2 925.203} C_VEL
LIN {X 0,Y 751.709,Z 809.06,A -85,B 0,C 180,E1 928.844,E2 928.844} C_VEL
LIN {X 0,Y 751.83,Z 809.06,A -85,B 0,C 180,E1 932.863,E2 932.863} C_VEL
LIN {X 0,Y 751.817,Z 809.06,A -85,B 0,C 180,E1 937.081,E2 937.081} C_VEL
LIN {X 0,Y 751.839,Z 809.06,A -85,B 0,C 180,E1 943.103,E2 943.103} C_VEL
LIN {X 0,Y 751.414,Z 809.06,A -85,B 0,C 180,E1 946.859,E2 946.859} C_VEL
LIN {X 0,Y 751.843,Z 809.06,A -85,B 0,C 180,E1 951.609,E2 951.609} C_VEL
LIN {X 0,Y 751.892,Z 809.06,A -85,B 0,C 180,E1 952.654,E2 952.654} C_VEL
LIN {X 0,Y 753.855,Z 816.996,A -85,B 0,C 180,E1 952.879,E2 952.879} C_VEL
LIN {X 0,Y 754.494,Z 921.374,A -85,B 0,C 180,E1 954.216,E2 954.216} C_VEL
LIN {X 0,Y 754.055,Z 966.455,A -85,B 0,C 180,E1 955.213,E2 955.213} C_VEL
LIN {X 0,Y 753.809,Z 1013.964,A -85,B 0,C 180,E1 956.774,E2 956.774} C_VEL
LIN {X 0,Y 753.387,Z 1061.185,A -85,B 0,C 180,E1 958.869,E2 958.869} C_VEL
LIN {X 0,Y 753.103,Z 1102.583,A -85,B 0,C 180,E1 961.208,E2 961.208} C_VEL
LIN {X 0,Y 752.644,Z 1144.367,A -85,B 0,C 180,E1 964.148,E2 964.148} C_VEL
LIN {X 0,Y 752.391,Z 1179.866,A -85,B 0,C 180,E1 967.252,E2 967.252} C_VEL
LIN {X 0,Y 752.105,Z 1209.891,A -85,B 0,C 180,E1 970.457,E2 970.457} C_VEL
LIN {X 0,Y 751.99,Z 1235.815,A -85,B 0,C 180,E1 973.946,E2 973.946} C_VEL
LIN {X 0,Y 751.872,Z 1256.534,A -85,B 0,C 180,E1 977.518,E2 977.518} C_VEL
LIN {X 0,Y 751.915,Z 1270.4,A -85,B 0,C 180,E1 980.744,E2 980.744} C_VEL
LIN {X 0,Y 751.958,Z 1280.559,A -85,B 0,C 180,E1 984.229,E2 984.229} C_VEL
LIN {X 0,Y 751.856,Z 1285.87,A -85,B 0,C 180,E1 987.692,E2 987.692} C_VEL
LIN {X 0,Y 751.985,Z 1286.67,A -85,B 0,C 180,E1 991.147,E2 991.147} C_VEL
LIN {X 0,Y 751.761,Z 1282.919,A -85,B 0,C 180,E1 994.607,E2 994.607} C_VEL
LIN {X 0,Y 751.711,Z 1274.303,A -85,B 0,C 180,E1 998.084,E2 998.084} C_VEL
LIN {X 0,Y 751.846,Z 1260.715,A -85,B 0,C 180,E1 1001.589,E2 1001.589} C_VEL
LIN {X 0,Y 751.886,Z 1243.49,A -85,B 0,C 180,E1 1004.842,E2 1004.842} C_VEL
LIN {X 0,Y 752.047,Z 1219.925,A -85,B 0,C 180,E1 1008.292,E2 1008.292} C_VEL
LIN {X 0,Y 752.238,Z 1189.311,A -85,B 0,C 180,E1 1011.81,E2 1011.81} C_VEL
LIN {X 0,Y 752.567,Z 1155.61,A -85,B 0,C 180,E1 1014.934,E2 1014.934} C_VEL
LIN {X 0,Y 752.943,Z 1116.034,A -85,B 0,C 180,E1 1017.92,E2 1017.92} C_VEL
LIN {X 0,Y 753.362,Z 1071.434,A -85,B 0,C 180,E1 1020.597,E2 1020.597} C_VEL
LIN {X 0,Y 753.818,Z 1028.97,A -85,B 0,C 180,E1 1022.618,E2 1022.618} C_VEL
LIN {X 0,Y 754.106,Z 983.592,A -85,B 0,C 180,E1 1024.27,E2 1024.27} C_VEL
LIN {X 0,Y 754.327,Z 940.929,A -85,B 0,C 180,E1 1025.405,E2 1025.405} C_VEL
LIN {X 0,Y 754.494,Z 896.697,A -85,B 0,C 180,E1 1026.154,E2 1026.154} C_VEL
LIN {X 0,Y 753.409,Z 813.776,A -85,B 0,C 180,E1 1027.184,E2 1027.184} C_VEL
LIN {X 0,Y 751.93,Z 809.06,A -85,B 0,C 180,E1 1027.333,E2 1027.333} C_VEL
LIN {X 0,Y 751.82,Z 809.06,A -85,B 0,C 180,E1 1033.654,E2 1033.654} C_VEL
LIN {X 0,Y 751.397,Z 809.06,A -85,B 0,C 180,E1 1038.424,E2 1038.424} C_VEL
LIN {X 0,Y 751.559,Z 809.06,A -85,B 0,C 180,E1 1041.631,E2 1041.631} C_VEL
LIN {X 0,Y 751.559,Z 809.06,A -85,B 0,C 180,E1 1045.741,E2 1045.741} C_VEL
LIN {X 0,Y 751.647,Z 809.06,A -85,B 0,C 180,E1 1049.83,E2 1049.83} C_VEL
LIN {X 0,Y 751.454,Z 809.06,A -85,B 0,C 180,E1 1055.022,E2 1055.022} C_VEL
LIN {X 0,Y 751.721,Z 809.06,A -85,B 0,C 180,E1 1060.019,E2 1060.019} C_VEL
LIN {X 0,Y 751.645,Z 809.06,A -85,B 0,C 180,E1 1066.04,E2 1066.04} C_VEL
LIN {X 0,Y 751.88,Z 809.847,A -85,B 0,C 180,E1 1069.874,E2 1069.874} C_VEL
LIN {X 0,Y 754.015,Z 818.22,A -85,B 0,C 180,E1 1070.216,E2 1070.216} C_VEL
LIN {X 0,Y 753.895,Z 865.376,A -85,B 0,C 180,E1 1071.79,E2 1071.79} C_VEL
LIN {X 0,Y 753.418,Z 911.461,A -85,B 0,C 180,E1 1073.839,E2 1073.839} C_VEL
LIN {X 0,Y 753.097,Z 952.983,A -85,B 0,C 180,E1 1076.189,E2 1076.189} C_VEL
LIN {X 0,Y 752.683,Z 994.799,A -85,B 0,C 180,E1 1079.137,E2 1079.137} C_VEL
LIN {X 0,Y 752.344,Z 1030.861,A -85,B 0,C 180,E1 1082.302,E2 1082.302} C_VEL
LIN {X 0,Y 752.199,Z 1061.536,A -85,B 0,C 180,E1 1085.619,E2 1085.619} C_VEL
LIN {X 0,Y 752,Z 1088.116,A -85,B 0,C 180,E1 1089.25,E2 1089.25} C_VEL
LIN {X 0,Y 751.995,Z 1107.964,A -85,B 0,C 180,E1 1092.769,E2 1092.769} C_VEL
LIN {X 0,Y 751.915,Z 1122.531,A -85,B 0,C 180,E1 1096.339,E2 1096.339} C_VEL
LIN {X 0,Y 751.947,Z 1132.201,A -85,B 0,C 180,E1 1099.974,E2 1099.974} C_VEL
LIN {X 0,Y 751.889,Z 1136.64,A -85,B 0,C 180,E1 1103.698,E2 1103.698} C_VEL
LIN {X 0,Y 751.862,Z 1135.637,A -85,B 0,C 180,E1 1107.53,E2 1107.53} C_VEL
LIN {X 0,Y 751.996,Z 1130.325,A -85,B 0,C 180,E1 1110.83,E2 1110.83} C_VEL
LIN {X 0,Y 752.026,Z 1119.121,A -85,B 0,C 180,E1 1114.54,E2 1114.54} C_VEL
LIN {X 0,Y 751.981,Z 1101.418,A -85,B 0,C 180,E1 1118.409,E2 1118.409} C_VEL
LIN {X 0,Y 752.068,Z 1079.193,A -85,B 0,C 180,E1 1121.985,E2 1121.985} C_VEL
LIN {X 0,Y 752.206,Z 1051.423,A -85,B 0,C 180,E1 1125.464,E2 1125.464} C_VEL
LIN {X 0,Y 752.463,Z 1019.531,A -85,B 0,C 180,E1 1128.675,E2 1128.675} C_VEL
LIN {X 0,Y 752.822,Z 981.917,A -85,B 0,C 180,E1 1131.754,E2 1131.754} C_VEL
LIN {X 0,Y 753.167,Z 940.271,A -85,B 0,C 180,E1 1134.493,E2 1134.493} C_VEL
LIN {X 0,Y 753.633,Z 897.269,A -85,B 0,C 180,E1 1136.764,E2 1136.764} C_VEL
LIN {X 0,Y 753.946,Z 851.226,A -85,B 0,C 180,E1 1138.642,E2 1138.642} C_VEL
LIN {X 0,Y 753.298,Z 813.579,A -85,B 0,C 180,E1 1139.862,E2 1139.862} C_VEL
LIN {X 0,Y 751.773,Z 809.06,A -85,B 0,C 180,E1 1140.078,E2 1140.078} C_VEL
LIN {X 0,Y 751.457,Z 809.06,A -85,B 0,C 180,E1 1145.027,E2 1145.027} C_VEL
LIN {X 0,Y 751.704,Z 809.06,A -85,B 0,C 180,E1 1150.023,E2 1150.023} C_VEL
LIN {X 0,Y 751.694,Z 809.06,A -85,B 0,C 180,E1 1156.046,E2 1156.046} C_VEL
LIN {X 0,Y 751.715,Z 809.06,A -85,B 0,C 180,E1 1160.751,E2 1160.751} C_VEL
LIN {X 0,Y 751.768,Z 809.06,A -85,B 0,C 180,E1 1164.237,E2 1164.237} C_VEL
LIN {X 0,Y 751.601,Z 809.06,A -85,B 0,C 180,E1 1168.853,E2 1168.853} C_VEL
LIN {X 0,Y 751.64,Z 809.06,A -85,B 0,C 180,E1 1172.309,E2 1172.309} C_VEL
LIN {X 0,Y 751.68,Z 809.06,A -85,B 0,C 180,E1 1175.773,E2 1175.773} C_VEL
LIN {X 0,Y 751.632,Z 809.06,A -85,B 0,C 180,E1 1180.429,E2 1180.429} C_VEL
LIN {X 0,Y 751.596,Z 809.06,A -85,B 0,C 180,E1 1183.965,E2 1183.965} C_VEL
LIN {X 0,Y 751.668,Z 809.06,A -85,B 0,C 180,E1 1187.555,E2 1187.555} C_VEL
LIN {X 0,Y 751.586,Z 809.06,A -85,B 0,C 180,E1 1191.221,E2 1191.221} C_VEL
LIN {X 0,Y 751.552,Z 809.06,A -85,B 0,C 180,E1 1195.215,E2 1195.215} C_VEL
LIN {X 0,Y 751.709,Z 809.06,A -85,B 0,C 180,E1 1198.85,E2 1198.85} C_VEL
LIN {X 0,Y 751.855,Z 809.06,A -85,B 0,C 180,E1 1202.869,E2 1202.869} C_VEL
LIN {X 0,Y 751.813,Z 809.06,A -85,B 0,C 180,E1 1207.088,E2 1207.088} C_VEL
LIN {X 0,Y 751.804,Z 809.06,A -85,B 0,C 180,E1 1213.113,E2 1213.113} C_VEL
LIN {X 0,Y 751.401,Z 809.06,A -85,B 0,C 180,E1 1216.867,E2 1216.867} C_VEL
LIN {X 0,Y 751.59,Z 809.06,A -85,B 0,C 180,E1 1221.449,E2 1221.449} C_VEL
LIN {X 0,Y 751.567,Z 809.06,A -85,B 0,C 180,E1 1225.742,E2 1225.742} C_VEL
LIN {X 0,Y 751.728,Z 809.06,A -85,B 0,C 180,E1 1229.835,E2 1229.835} C_VEL
LIN {X 0,Y 751.707,Z 809.06,A -85,B 0,C 180,E1 1234.776,E2 1234.776} C_VEL
LIN {X 0,Y 751.702,Z 809.06,A -85,B 0,C 180,E1 1238.789,E2 1238.789} C_VEL
LIN {X 0,Y 751.705,Z 809.06,A -85,B 0,C 180,E1 1243.656,E2 1243.656} C_VEL
LIN {X 0,Y 751.59,Z 809.06,A -85,B 0,C 180,E1 1248.403,E2 1248.403} C_VEL
LIN {X 0,Y 751.663,Z 809.06,A -85,B 0,C 180,E1 1251.911,E2 1251.911} C_VEL
LIN {X 0,Y 751.836,Z 809.06,A -85,B 0,C 180,E1 1256.544,E2 1256.544} C_VEL
LIN {X 0,Y 751.716,Z 809.06,A -85,B 0,C 180,E1 1258.321,E2 1258.321} C_VEL
LIN {X 0,Y 747.74,Z 809.06,A -85,B 0,C 180,E1 1259.627,E2 1259.627} C_VEL
LIN {X 0,Y 744.042,Z 809.06,A -85,B 0,C 180,E1 1260.947,E2 1260.947} C_VEL
LIN {X 0,Y 743.855,Z 809.06,A -85,B 0,C 180,E1 1265.83,E2 1265.83} C_VEL
LIN {X 0,Y 743.74,Z 809.06,A -85,B 0,C 180,E1 1270.536,E2 1270.536} C_VEL
LIN {X 0,Y 743.843,Z 809.06,A -85,B 0,C 180,E1 1275.312,E2 1275.312} C_VEL
LIN {X 0,Y 743.863,Z 809.06,A -85,B 0,C 180,E1 1280.202,E2 1280.202} C_VEL
LIN {X 0,Y 743.674,Z 809.06,A -85,B 0,C 180,E1 1285.257,E2 1285.257} C_VEL
LIN {X 0,Y 743.724,Z 809.06,A -85,B 0,C 180,E1 1289.183,E2 1289.183} C_VEL
LIN {X 0,Y 743.748,Z 809.06,A -85,B 0,C 180,E1 1293.585,E2 1293.585} C_VEL
LIN {X 0,Y 743.752,Z 809.06,A -85,B 0,C 180,E1 1297.587,E2 1297.587} C_VEL
LIN {X 0,Y 743.917,Z 809.06,A -85,B 0,C 180,E1 1303.003,E2 1303.003} C_VEL
LIN {X 0,Y 743.513,Z 809.06,A -85,B 0,C 180,E1 1307.022,E2 1307.022} C_VEL
LIN {X 0,Y 743.945,Z 809.06,A -85,B 0,C 180,E1 1312.177,E2 1312.177} C_VEL
LIN {X 0,Y 747.598,Z 818.931,A -85,B 0,C 180,E1 1312.538,E2 1312.538} C_VEL
LIN {X 0,Y 748.067,Z 921.576,A -85,B 0,C 180,E1 1313.865,E2 1313.865} C_VEL
LIN {X 0,Y 747.495,Z 965.992,A -85,B 0,C 180,E1 1314.85,E2 1314.85} C_VEL
LIN {X 0,Y 747.02,Z 1014.046,A -85,B 0,C 180,E1 1316.436,E2 1316.436} C_VEL
LIN {X 0,Y 746.336,Z 1062.43,A -85,B 0,C 180,E1 1318.604,E2 1318.604} C_VEL
LIN {X 0,Y 745.827,Z 1104.107,A -85,B 0,C 180,E1 1321.002,E2 1321.002} C_VEL
LIN {X 0,Y 745.218,Z 1145.116,A -85,B 0,C 180,E1 1323.929,E2 1323.929} C_VEL
LIN {X 0,Y 744.759,Z 1181.474,A -85,B 0,C 180,E1 1327.163,E2 1327.163} C_VEL
LIN {X 0,Y 744.356,Z 1211.052,A -85,B 0,C 180,E1 1330.391,E2 1330.391} C_VEL
LIN {X 0,Y 744.129,Z 1237.859,A -85,B 0,C 180,E1 1334.085,E2 1334.085} C_VEL
LIN {X 0,Y 744.025,Z 1256.586,A -85,B 0,C 180,E1 1337.395,E2 1337.395} C_VEL
LIN {X 0,Y 744.043,Z 1270.4,A -85,B 0,C 180,E1 1340.645,E2 1340.645} C_VEL
LIN {X 0,Y 744.059,Z 1280.871,A -85,B 0,C 180,E1 1344.308,E2 1344.308} C_VEL
LIN {X 0,Y 743.953,Z 1285.87,A -85,B 0,C 180,E1 1347.667,E2 1347.667} C_VEL
LIN {X 0,Y 744.084,Z 1286.67,A -85,B 0,C 180,E1 1351.159,E2 1351.159} C_VEL
LIN {X 0,Y 743.86,Z 1282.919,A -85,B 0,C 180,E1 1354.656,E2 1354.656} C_VEL
LIN {X 0,Y 743.91,Z 1276.115,A -85,B 0,C 180,E1 1357.582,E2 1357.582} C_VEL
LIN {X 0,Y 744.069,Z 1263.417,A -85,B 0,C 180,E1 1361.119,E2 1361.119} C_VEL
LIN {X 0,Y 744.061,Z 1245.25,A -85,B 0,C 180,E1 1364.701,E2 1364.701} C_VEL
LIN {X 0,Y 744.275,Z 1222.208,A -85,B 0,C 180,E1 1368.184,E2 1368.184} C_VEL
LIN {X 0,Y 744.573,Z 1193.788,A -85,B 0,C 180,E1 1371.571,E2 1371.571} C_VEL
LIN {X 0,Y 745.055,Z 1159.26,A -85,B 0,C 180,E1 1374.897,E2 1374.897} C_VEL
LIN {X 0,Y 745.604,Z 1118.407,A -85,B 0,C 180,E1 1378.051,E2 1378.051} C_VEL
LIN {X 0,Y 746.2,Z 1076.649,A -85,B 0,C 180,E1 1380.632,E2 1380.632} C_VEL
LIN {X 0,Y 746.877,Z 1032.998,A -85,B 0,C 180,E1 1382.783,E2 1382.783} C_VEL
LIN {X 0,Y 747.41,Z 988.278,A -85,B 0,C 180,E1 1384.471,E2 1384.471} C_VEL
LIN {X 0,Y 747.808,Z 943.218,A -85,B 0,C 180,E1 1385.709,E2 1385.709} C_VEL
LIN {X 0,Y 748.122,Z 899.326,A -85,B 0,C 180,E1 1386.478,E2 1386.478} C_VEL
LIN {X 0,Y 747.271,Z 817.141,A -85,B 0,C 180,E1 1387.502,E2 1387.502} C_VEL
LIN {X 0,Y 743.789,Z 809.06,A -85,B 0,C 180,E1 1387.85,E2 1387.85} C_VEL
LIN {X 0,Y 743.918,Z 809.06,A -85,B 0,C 180,E1 1393.672,E2 1393.672} C_VEL
LIN {X 0,Y 743.528,Z 809.06,A -85,B 0,C 180,E1 1398.751,E2 1398.751} C_VEL
LIN {X 0,Y 743.536,Z 809.06,A -85,B 0,C 180,E1 1402.435,E2 1402.435} C_VEL
LIN {X 0,Y 743.511,Z 809.06,A -85,B 0,C 180,E1 1406.721,E2 1406.721} C_VEL
LIN {X 0,Y 743.559,Z 809.06,A -85,B 0,C 180,E1 1410.898,E2 1410.898} C_VEL
LIN {X 0,Y 743.633,Z 809.06,A -85,B 0,C 180,E1 1414.741,E2 1414.741} C_VEL
LIN {X 0,Y 743.738,Z 809.06,A -85,B 0,C 180,E1 1419.795,E2 1419.795} C_VEL
LIN {X 0,Y 743.707,Z 809.06,A -85,B 0,C 180,E1 1425.888,E2 1425.888} C_VEL
LIN {X 0,Y 743.797,Z 809.556,A -85,B 0,C 180,E1 1429.428,E2 1429.428} C_VEL
LIN {X 0,Y 747.403,Z 820.147,A -85,B 0,C 180,E1 1429.918,E2 1429.918} C_VEL
LIN {X 0,Y 747.1,Z 866.515,A -85,B 0,C 180,E1 1431.495,E2 1431.495} C_VEL
LIN {X 0,Y 746.417,Z 911.934,A -85,B 0,C 180,E1 1433.538,E2 1433.538} C_VEL
LIN {X 0,Y 745.834,Z 953.764,A -85,B 0,C 180,E1 1435.933,E2 1435.933} C_VEL
LIN {X 0,Y 745.245,Z 994.517,A -85,B 0,C 180,E1 1438.838,E2 1438.838} C_VEL
LIN {X 0,Y 744.709,Z 1030.641,A -85,B 0,C 180,E1 1442.034,E2 1442.034} C_VEL
LIN {X 0,Y 744.46,Z 1061.348,A -85,B 0,C 180,E1 1445.386,E2 1445.386} C_VEL
LIN {X 0,Y 744.135,Z 1087.95,A -85,B 0,C 180,E1 1449.054,E2 1449.054} C_VEL
LIN {X 0,Y 744.116,Z 1107.831,A -85,B 0,C 180,E1 1452.608,E2 1452.608} C_VEL
LIN {X 0,Y 744.032,Z 1123.423,A -85,B 0,C 180,E1 1456.517,E2 1456.517} C_VEL
LIN {X 0,Y 744.017,Z 1132.73,A -85,B 0,C 180,E1 1460.196,E2 1460.196} C_VEL
LIN {X 0,Y 743.949,Z 1136.724,A -85,B 0,C 180,E1 1463.966,E2 1463.966} C_VEL
LIN {X 0,Y 743.929,Z 1135.385,A -85,B 0,C 180,E1 1467.849,E2 1467.849} C_VEL
LIN {X 0,Y 743.992,Z 1128.974,A -85,B 0,C 180,E1 1471.468,E2 1471.468} C_VEL
LIN {X 0,Y 743.999,Z 1117.862,A -85,B 0,C 180,E1 1474.967,E2 1474.967} C_VEL
LIN {X 0,Y 744.107,Z 1101.051,A -85,B 0,C 180,E1 1478.626,E2 1478.626} C_VEL
LIN {X 0,Y 744.249,Z 1079.956,A -85,B 0,C 180,E1 1482.064,E2 1482.064} C_VEL
LIN {X 0,Y 744.488,Z 1050.917,A -85,B 0,C 180,E1 1485.746,E2 1485.746} C_VEL
LIN {X 0,Y 744.866,Z 1019.537,A -85,B 0,C 180,E1 1488.932,E2 1488.932} C_VEL
LIN {X 0,Y 745.393,Z 982.061,A -85,B 0,C 180,E1 1492.032,E2 1492.032} C_VEL
LIN {X 0,Y 745.977,Z 941.465,A -85,B 0,C 180,E1 1494.734,E2 1494.734} C_VEL
LIN {X 0,Y 746.675,Z 898.084,A -85,B 0,C 180,E1 1497.058,E2 1497.058} C_VEL
LIN {X 0,Y 747.233,Z 852.044,A -85,B 0,C 180,E1 1498.956,E2 1498.956} C_VEL
LIN {X 0,Y 746.715,Z 817.06,A -85,B 0,C 180,E1 1500.117,E2 1500.117} C_VEL
LIN {X 0,Y 743.699,Z 809.06,A -85,B 0,C 180,E1 1500.57,E2 1500.57} C_VEL
LIN {X 0,Y 743.637,Z 809.06,A -85,B 0,C 180,E1 1504.746,E2 1504.746} C_VEL
LIN {X 0,Y 743.723,Z 809.06,A -85,B 0,C 180,E1 1509.799,E2 1509.799} C_VEL
LIN {X 0,Y 743.75,Z 809.06,A -85,B 0,C 180,E1 1515.894,E2 1515.894} C_VEL
LIN {X 0,Y 743.856,Z 809.06,A -85,B 0,C 180,E1 1520.652,E2 1520.652} C_VEL
LIN {X 0,Y 743.83,Z 809.06,A -85,B 0,C 180,E1 1524.478,E2 1524.478} C_VEL
LIN {X 0,Y 743.703,Z 809.06,A -85,B 0,C 180,E1 1528.841,E2 1528.841} C_VEL
LIN {X 0,Y 743.738,Z 809.06,A -85,B 0,C 180,E1 1532.334,E2 1532.334} C_VEL
LIN {X 0,Y 743.785,Z 809.06,A -85,B 0,C 180,E1 1535.835,E2 1535.835} C_VEL
LIN {X 0,Y 743.732,Z 809.06,A -85,B 0,C 180,E1 1540.541,E2 1540.541} C_VEL
LIN {X 0,Y 743.846,Z 809.06,A -85,B 0,C 180,E1 1545.317,E2 1545.317} C_VEL
LIN {X 0,Y 743.87,Z 809.06,A -85,B 0,C 180,E1 1550.207,E2 1550.207} C_VEL
LIN {X 0,Y 743.674,Z 809.06,A -85,B 0,C 180,E1 1555.263,E2 1555.263} C_VEL
LIN {X 0,Y 743.747,Z 809.06,A -85,B 0,C 180,E1 1559.188,E2 1559.188} C_VEL
LIN {X 0,Y 743.763,Z 809.06,A -85,B 0,C 180,E1 1563.6,E2 1563.6} C_VEL
LIN {X 0,Y 743.749,Z 809.06,A -85,B 0,C 180,E1 1567.598,E2 1567.598} C_VEL
LIN {X 0,Y 743.9,Z 809.06,A -85,B 0,C 180,E1 1573.686,E2 1573.686} C_VEL
LIN {X 0,Y 743.5,Z 809.06,A -85,B 0,C 180,E1 1578.768,E2 1578.768} C_VEL
LIN {X 0,Y 743.524,Z 809.06,A -85,B 0,C 180,E1 1582.436,E2 1582.436} C_VEL
LIN {X 0,Y 743.531,Z 809.06,A -85,B 0,C 180,E1 1586.723,E2 1586.723} C_VEL
LIN {X 0,Y 743.679,Z 809.06,A -85,B 0,C 180,E1 1590.901,E2 1590.901} C_VEL
LIN {X 0,Y 743.84,Z 809.06,A -85,B 0,C 180,E1 1594.75,E2 1594.75} C_VEL
LIN {X 0,Y 743.753,Z 809.06,A -85,B 0,C 180,E1 1599.17,E2 1599.17} C_VEL
LIN {X 0,Y 743.801,Z 809.06,A -85,B 0,C 180,E1 1603.477,E2 1603.477} C_VEL
LIN {X 0,Y 743.669,Z 809.06,A -85,B 0,C 180,E1 1608.277,E2 1608.277} C_VEL
LIN {X 0,Y 743.983,Z 809.06,A -85,B 0,C 180,E1 1613.149,E2 1613.149} C_VEL
LIN {X 0,Y 743.813,Z 809.06,A -85,B 0,C 180,E1 1618.313,E2 1618.313} C_VEL
LIN {X 0,Y 744.042,Z 809.06,A -85,B 0,C 180,E1 1620.947,E2 1620.947} C_VEL
LIN {X 0,Y 741.562,Z 809.06,A -85,B 0,C 180,E1 1621.938,E2 1621.938} C_VEL
LIN {X 0,Y 736.049,Z 809.06,A -85,B 0,C 180,E1 1623.415,E2 1623.415} C_VEL
LIN {X 0,Y 735.961,Z 809.06,A -85,B 0,C 180,E1 1623.586,E2 1623.586} C_VEL
LIN {X 0,Y 736.044,Z 809.06,A -85,B 0,C 180,E1 1628.262,E2 1628.262} C_VEL
LIN {X 0,Y 735.944,Z 809.06,A -85,B 0,C 180,E1 1633.053,E2 1633.053} C_VEL
LIN {X 0,Y 735.818,Z 809.06,A -85,B 0,C 180,E1 1637.941,E2 1637.941} C_VEL
LIN {X 0,Y 735.731,Z 809.06,A -85,B 0,C 180,E1 1642.438,E2 1642.438} C_VEL
LIN {X 0,Y 735.713,Z 809.06,A -85,B 0,C 180,E1 1646.862,E2 1646.862} C_VEL
LIN {X 0,Y 735.891,Z 809.06,A -85,B 0,C 180,E1 1652.267,E2 1652.267} C_VEL
LIN {X 0,Y 735.793,Z 809.06,A -85,B 0,C 180,E1 1656.775,E2 1656.775} C_VEL
LIN {X 0,Y 735.963,Z 809.06,A -85,B 0,C 180,E1 1662.65,E2 1662.65} C_VEL
LIN {X 0,Y 735.576,Z 809.06,A -85,B 0,C 180,E1 1667.314,E2 1667.314} C_VEL
LIN {X 0,Y 736.027,Z 809.06,A -85,B 0,C 180,E1 1671.724,E2 1671.724} C_VEL
LIN {X 0,Y 740.694,Z 819.323,A -85,B 0,C 180,E1 1672.133,E2 1672.133} C_VEL
LIN {X 0,Y 741.739,Z 845.705,A -85,B 0,C 180,E1 1672.511,E2 1672.511} C_VEL
LIN {X 0,Y 741.678,Z 921.558,A -85,B 0,C 180,E1 1673.503,E2 1673.503} C_VEL
LIN {X 0,Y 740.978,Z 965.549,A -85,B 0,C 180,E1 1674.481,E2 1674.481} C_VEL
LIN {X 0,Y 740.283,Z 1014.042,A -85,B 0,C 180,E1 1676.089,E2 1676.089} C_VEL
LIN {X 0,Y 739.339,Z 1062.438,A -85,B 0,C 180,E1 1678.273,E2 1678.273} C_VEL
LIN {X 0,Y 738.587,Z 1104.863,A -85,B 0,C 180,E1 1680.741,E2 1680.741} C_VEL
LIN {X 0,Y 737.758,Z 1145.665,A -85,B 0,C 180,E1 1683.688,E2 1683.688} C_VEL
LIN {X 0,Y 737.139,Z 1183.088,A -85,B 0,C 180,E1 1687.073,E2 1687.073} C_VEL
LIN {X 0,Y 736.576,Z 1213.46,A -85,B 0,C 180,E1 1690.484,E2 1690.484} C_VEL
LIN {X 0,Y 736.33,Z 1237.861,A -85,B 0,C 180,E1 1693.912,E2 1693.912} C_VEL
LIN {X 0,Y 736.182,Z 1256.686,A -85,B 0,C 180,E1 1697.278,E2 1697.278} C_VEL
LIN {X 0,Y 736.172,Z 1270.4,A -85,B 0,C 180,E1 1700.544,E2 1700.544} C_VEL
LIN {X 0,Y 736.103,Z 1281.436,A -85,B 0,C 180,E1 1704.511,E2 1704.511} C_VEL
LIN {X 0,Y 736.059,Z 1285.87,A -85,B 0,C 180,E1 1707.642,E2 1707.642} C_VEL
LIN {X 0,Y 736.19,Z 1286.67,A -85,B 0,C 180,E1 1711.171,E2 1711.171} C_VEL
LIN {X 0,Y 735.974,Z 1282.919,A -85,B 0,C 180,E1 1714.706,E2 1714.706} C_VEL
LIN {X 0,Y 736.016,Z 1276.116,A -85,B 0,C 180,E1 1717.664,E2 1717.664} C_VEL
LIN {X 0,Y 736.174,Z 1263.418,A -85,B 0,C 180,E1 1721.239,E2 1721.239} C_VEL
LIN {X 0,Y 736.205,Z 1244.32,A -85,B 0,C 180,E1 1725.022,E2 1725.022} C_VEL
LIN {X 0,Y 736.496,Z 1221.108,A -85,B 0,C 180,E1 1728.537,E2 1728.537} C_VEL
LIN {X 0,Y 736.912,Z 1192.789,A -85,B 0,C 180,E1 1731.914,E2 1731.914} C_VEL
LIN {X 0,Y 737.542,Z 1159.443,A -85,B 0,C 180,E1 1735.153,E2 1735.153} C_VEL
LIN {X 0,Y 738.288,Z 1118.434,A -85,B 0,C 180,E1 1738.352,E2 1738.352} C_VEL
LIN {X 0,Y 739.099,Z 1077.659,A -85,B 0,C 180,E1 1740.902,E2 1740.902} C_VEL
LIN {X 0,Y 740.011,Z 1034.096,A -85,B 0,C 180,E1 1743.075,E2 1743.075} C_VEL
LIN {X 0,Y 740.753,Z 990.295,A -85,B 0,C 180,E1 1744.761,E2 1744.761} C_VEL
LIN {X 0,Y 741.314,Z 944.588,A -85,B 0,C 180,E1 1746.039,E2 1746.039} C_VEL
LIN {X 0,Y 741.747,Z 900.422,A -85,B 0,C 180,E1 1746.828,E2 1746.828} C_VEL
LIN {X 0,Y 740.877,Z 819.648,A -85,B 0,C 180,E1 1747.853,E2 1747.853} C_VEL
LIN {X 0,Y 735.81,Z 810.151,A -85,B 0,C 180,E1 1748.275,E2 1748.275} C_VEL
LIN {X 0,Y 735.749,Z 809.06,A -85,B 0,C 180,E1 1748.299,E2 1748.299} C_VEL
LIN {X 0,Y 736.016,Z 809.06,A -85,B 0,C 180,E1 1754.067,E2 1754.067} C_VEL
LIN {X 0,Y 735.801,Z 809.06,A -85,B 0,C 180,E1 1759.442,E2 1759.442} C_VEL
LIN {X 0,Y 735.793,Z 809.06,A -85,B 0,C 180,E1 1765.222,E2 1765.222} C_VEL
LIN {X 0,Y 735.675,Z 809.06,A -85,B 0,C 180,E1 1770.466,E2 1770.466} C_VEL
LIN {X 0,Y 735.732,Z 809.06,A -85,B 0,C 180,E1 1774.634,E2 1774.634} C_VEL
LIN {X 0,Y 735.786,Z 809.06,A -85,B 0,C 180,E1 1779.567,E2 1779.567} C_VEL
LIN {X 0,Y 735.771,Z 809.06,A -85,B 0,C 180,E1 1785.733,E2 1785.733} C_VEL
LIN {X 0,Y 735.758,Z 809.436,A -85,B 0,C 180,E1 1788.976,E2 1788.976} C_VEL
LIN {X 0,Y 740.826,Z 822.569,A -85,B 0,C 180,E1 1789.631,E2 1789.631} C_VEL
LIN {X 0,Y 740.196,Z 871.333,A -85,B 0,C 180,E1 1791.341,E2 1791.341} C_VEL
LIN {X 0,Y 739.308,Z 917.228,A -85,B 0,C 180,E1 1793.475,E2 1793.475} C_VEL
LIN {X 0,Y 738.459,Z 961.195,A -85,B 0,C 180,E1 1796.113,E2 1796.113} C_VEL
LIN {X 0,Y 737.714,Z 999.606,A -85,B 0,C 180,E1 1798.973,E2 1798.973} C_VEL
LIN {X 0,Y 737.073,Z 1034.875,A -85,B 0,C 180,E1 1802.202,E2 1802.202} C_VEL
LIN {X 0,Y 736.67,Z 1064.403,A -85,B 0,C 180,E1 1805.561,E2 1805.561} C_VEL
LIN {X 0,Y 736.35,Z 1089.69,A -85,B 0,C 180,E1 1809.15,E2 1809.15} C_VEL
LIN {X 0,Y 736.254,Z 1108.967,A -85,B 0,C 180,E1 1812.727,E2 1812.727} C_VEL
LIN {X 0,Y 736.181,Z 1124.312,A -85,B 0,C 180,E1 1816.699,E2 1816.699} C_VEL
LIN {X 0,Y 736.085,Z 1133.194,A -85,B 0,C 180,E1 1820.424,E2 1820.424} C_VEL
LIN {X 0,Y 736,Z 1136.808,A -85,B 0,C 180,E1 1824.242,E2 1824.242} C_VEL
LIN {X 0,Y 735.992,Z 1135.084,A -85,B 0,C 180,E1 1828.176,E2 1828.176} C_VEL
LIN {X 0,Y 736.035,Z 1128.313,A -85,B 0,C 180,E1 1831.804,E2 1831.804} C_VEL
LIN {X 0,Y 736.124,Z 1117.843,A -85,B 0,C 180,E1 1835.081,E2 1835.081} C_VEL
LIN {X 0,Y 736.219,Z 1101.163,A -85,B 0,C 180,E1 1838.754,E2 1838.754} C_VEL
LIN {X 0,Y 736.415,Z 1078.987,A -85,B 0,C 180,E1 1842.388,E2 1842.388} C_VEL
LIN {X 0,Y 736.781,Z 1051.21,A -85,B 0,C 180,E1 1845.939,E2 1845.939} C_VEL
LIN {X 0,Y 737.291,Z 1019.362,A -85,B 0,C 180,E1 1849.21,E2 1849.21} C_VEL
LIN {X 0,Y 738.045,Z 981.655,A -85,B 0,C 180,E1 1852.354,E2 1852.354} C_VEL
LIN {X 0,Y 738.845,Z 939.849,A -85,B 0,C 180,E1 1855.151,E2 1855.151} C_VEL
LIN {X 0,Y 739.784,Z 897.387,A -85,B 0,C 180,E1 1857.427,E2 1857.427} C_VEL
LIN {X 0,Y 740.521,Z 852.931,A -85,B 0,C 180,E1 1859.275,E2 1859.275} C_VEL
LIN {X 0,Y 740.234,Z 820.353,A -85,B 0,C 180,E1 1860.377,E2 1860.377} C_VEL
LIN {X 0,Y 735.711,Z 809.06,A -85,B 0,C 180,E1 1861.026,E2 1861.026} C_VEL
LIN {X 0,Y 735.551,Z 809.06,A -85,B 0,C 180,E1 1865.746,E2 1865.746} C_VEL
LIN {X 0,Y 735.7,Z 809.06,A -85,B 0,C 180,E1 1870.864,E2 1870.864} C_VEL
LIN {X 0,Y 735.809,Z 809.06,A -85,B 0,C 180,E1 1875.739,E2 1875.739} C_VEL
LIN {X 0,Y 735.963,Z 809.06,A -85,B 0,C 180,E1 1880.551,E2 1880.551} C_VEL
LIN {X 0,Y 735.866,Z 809.06,A -85,B 0,C 180,E1 1885.293,E2 1885.293} C_VEL
LIN {X 0,Y 735.908,Z 809.06,A -85,B 0,C 180,E1 1890.005,E2 1890.005} C_VEL
LIN {X 0,Y 736.123,Z 809.06,A -85,B 0,C 180,E1 1894.715,E2 1894.715} C_VEL
LIN {X 0,Y 735.88,Z 809.06,A -85,B 0,C 180,E1 1899.742,E2 1899.742} C_VEL
LIN {X 0,Y 735.794,Z 809.06,A -85,B 0,C 180,E1 1904.272,E2 1904.272} C_VEL
LIN {X 0,Y 735.849,Z 809.06,A -85,B 0,C 180,E1 1907.945,E2 1907.945} C_VEL
LIN {X 0,Y 735.833,Z 809.06,A -85,B 0,C 180,E1 1912.97,E2 1912.97} C_VEL
LIN {X 0,Y 735.866,Z 809.06,A -85,B 0,C 180,E1 1918.188,E2 1918.188} C_VEL
LIN {X 0,Y 735.844,Z 809.06,A -85,B 0,C 180,E1 1923.678,E2 1923.678} C_VEL
LIN {X 0,Y 735.576,Z 809.06,A -85,B 0,C 180,E1 1928.687,E2 1928.687} C_VEL
LIN {X 0,Y 735.992,Z 809.06,A -85,B 0,C 180,E1 1934.066,E2 1934.066} C_VEL
LIN {X 0,Y 735.754,Z 809.06,A -85,B 0,C 180,E1 1939.461,E2 1939.461} C_VEL
LIN {X 0,Y 735.775,Z 809.06,A -85,B 0,C 180,E1 1945.241,E2 1945.241} C_VEL
LIN {X 0,Y 735.779,Z 809.06,A -85,B 0,C 180,E1 1950.472,E2 1950.472} C_VEL
LIN {X 0,Y 735.936,Z 809.06,A -85,B 0,C 180,E1 1954.623,E2 1954.623} C_VEL
LIN {X 0,Y 735.814,Z 809.06,A -85,B 0,C 180,E1 1959.569,E2 1959.569} C_VEL
LIN {X 0,Y 735.893,Z 809.06,A -85,B 0,C 180,E1 1964.519,E2 1964.519} C_VEL
LIN {X 0,Y 735.978,Z 809.06,A -85,B 0,C 180,E1 1970.257,E2 1970.257} C_VEL
LIN {X 0,Y 735.992,Z 809.06,A -85,B 0,C 180,E1 1974.109,E2 1974.109} C_VEL
LIN {X 0,Y 735.895,Z 809.06,A -85,B 0,C 180,E1 1978.824,E2 1978.824} C_VEL
LIN {X 0,Y 735.934,Z 809.06,A -85,B 0,C 180,E1 1982.354,E2 1982.354} C_VEL
LIN {X 0,Y 735.961,Z 809.06,A -85,B 0,C 180,E1 1983.586,E2 1983.586} C_VEL
LIN {X 0,Y 734.74,Z 809.06,A -85,B 0,C 180,E1 1984.261,E2 1984.261} C_VEL
LIN {X 0,Y 728.12,Z 809.06,A -85,B 0,C 180,E1 1986.092,E2 1986.092} C_VEL
LIN {X 0,Y 728.012,Z 809.06,A -85,B 0,C 180,E1 1986.265,E2 1986.265} C_VEL
LIN {X 0,Y 727.949,Z 809.06,A -85,B 0,C 180,E1 1990.767,E2 1990.767} C_VEL
LIN {X 0,Y 728.052,Z 809.06,A -85,B 0,C 180,E1 1995.653,E2 1995.653} C_VEL
LIN {X 0,Y 727.926,Z 809.06,A -85,B 0,C 180,E1 2000.9,E2 2000.9} C_VEL
LIN {X 0,Y 727.796,Z 809.06,A -85,B 0,C 180,E1 2005.848,E2 2005.848} C_VEL
LIN {X 0,Y 727.839,Z 809.06,A -85,B 0,C 180,E1 2009.884,E2 2009.884} C_VEL
LIN {X 0,Y 727.858,Z 809.06,A -85,B 0,C 180,E1 2014.091,E2 2014.091} C_VEL
LIN {X 0,Y 727.713,Z 809.06,A -85,B 0,C 180,E1 2018.529,E2 2018.529} C_VEL
LIN {X 0,Y 728.037,Z 809.06,A -85,B 0,C 180,E1 2023.405,E2 2023.405} C_VEL
LIN {X 0,Y 727.686,Z 809.06,A -85,B 0,C 180,E1 2028.376,E2 2028.376} C_VEL
LIN {X 0,Y 728.138,Z 809.794,A -85,B 0,C 180,E1 2031.242,E2 2031.242} C_VEL
LIN {X 0,Y 735.197,Z 824.11,A -85,B 0,C 180,E1 2031.857,E2 2031.857} C_VEL
LIN {X 0,Y 735.322,Z 920.656,A -85,B 0,C 180,E1 2033.12,E2 2033.12} C_VEL
LIN {X 0,Y 734.476,Z 964.068,A -85,B 0,C 180,E1 2034.077,E2 2034.077} C_VEL
LIN {X 0,Y 733.581,Z 1012.829,A -85,B 0,C 180,E1 2035.686,E2 2035.686} C_VEL
LIN {X 0,Y 732.368,Z 1060.834,A -85,B 0,C 180,E1 2037.852,E2 2037.852} C_VEL
LIN {X 0,Y 731.413,Z 1103.614,A -85,B 0,C 180,E1 2040.34,E2 2040.34} C_VEL
LIN {X 0,Y 730.344,Z 1145.872,A -85,B 0,C 180,E1 2043.417,E2 2043.417} C_VEL
LIN {X 0,Y 729.518,Z 1183.089,A -85,B 0,C 180,E1 2046.819,E2 2046.819} C_VEL
LIN {X 0,Y 728.863,Z 1212.544,A -85,B 0,C 180,E1 2050.15,E2 2050.15} C_VEL
LIN {X 0,Y 728.533,Z 1237.863,A -85,B 0,C 180,E1 2053.735,E2 2053.735} C_VEL
LIN {X 0,Y 728.319,Z 1256.906,A -85,B 0,C 180,E1 2057.182,E2 2057.182} C_VEL
LIN {X 0,Y 728.175,Z 1272.338,A -85,B 0,C 180,E1 2061.042,E2 2061.042} C_VEL
LIN {X 0,Y 728.28,Z 1280.559,A -85,B 0,C 180,E1 2064.041,E2 2064.041} C_VEL
LIN {X 0,Y 728.156,Z 1285.87,A -85,B 0,C 180,E1 2067.616,E2 2067.616} C_VEL
LIN {X 0,Y 728.288,Z 1286.67,A -85,B 0,C 180,E1 2071.184,E2 2071.184} C_VEL
LIN {X 0,Y 728.071,Z 1282.437,A -85,B 0,C 180,E1 2075.018,E2 2075.018} C_VEL
LIN {X 0,Y 728.019,Z 1274.305,A -85,B 0,C 180,E1 2078.349,E2 2078.349} C_VEL
LIN {X 0,Y 728.263,Z 1262.069,A -85,B 0,C 180,E1 2081.666,E2 2081.666} C_VEL
LIN {X 0,Y 728.368,Z 1243.371,A -85,B 0,C 180,E1 2085.354,E2 2085.354} C_VEL
LIN {X 0,Y 728.723,Z 1221.108,A -85,B 0,C 180,E1 2088.743,E2 2088.743} C_VEL
LIN {X 0,Y 729.235,Z 1191.964,A -85,B 0,C 180,E1 2092.247,E2 2092.247} C_VEL
LIN {X 0,Y 730.03,Z 1159.442,A -85,B 0,C 180,E1 2095.43,E2 2095.43} C_VEL
LIN {X 0,Y 731.044,Z 1118.433,A -85,B 0,C 180,E1 2098.658,E2 2098.658} C_VEL
LIN {X 0,Y 732.093,Z 1077.153,A -85,B 0,C 180,E1 2101.26,E2 2101.26} C_VEL
LIN {X 0,Y 733.211,Z 1033.216,A -85,B 0,C 180,E1 2103.463,E2 2103.463} C_VEL
LIN {X 0,Y 734.155,Z 990.23,A -85,B 0,C 180,E1 2105.121,E2 2105.121} C_VEL
LIN {X 0,Y 734.875,Z 945.064,A -85,B 0,C 180,E1 2106.394,E2 2106.394} C_VEL
LIN {X 0,Y 735.433,Z 899.928,A -85,B 0,C 180,E1 2107.204,E2 2107.204} C_VEL
LIN {X 0,Y 734.576,Z 823.035,A -85,B 0,C 180,E1 2108.194,E2 2108.194} C_VEL
LIN {X 0,Y 727.817,Z 810.108,A -85,B 0,C 180,E1 2108.774,E2 2108.774} C_VEL
LIN {X 0,Y 727.768,Z 809.06,A -85,B 0,C 180,E1 2108.8,E2 2108.8} C_VEL
LIN {X 0,Y 728.035,Z 809.06,A -85,B 0,C 180,E1 2113.414,E2 2113.414} C_VEL
LIN {X 0,Y 727.721,Z 809.06,A -85,B 0,C 180,E1 2118.367,E2 2118.367} C_VEL
LIN {X 0,Y 727.738,Z 809.06,A -85,B 0,C 180,E1 2122.977,E2 2122.977} C_VEL
LIN {X 0,Y 727.688,Z 809.06,A -85,B 0,C 180,E1 2127.325,E2 2127.325} C_VEL
LIN {X 0,Y 727.681,Z 809.06,A -85,B 0,C 180,E1 2131.472,E2 2131.472} C_VEL
LIN {X 0,Y 727.618,Z 809.06,A -85,B 0,C 180,E1 2136.017,E2 2136.017} C_VEL
LIN {X 0,Y 727.797,Z 809.06,A -85,B 0,C 180,E1 2140.599,E2 2140.599} C_VEL
LIN {X 0,Y 727.856,Z 809.06,A -85,B 0,C 180,E1 2145.575,E2 2145.575} C_VEL
LIN {X 0,Y 727.76,Z 809.157,A -85,B 0,C 180,E1 2148.51,E2 2148.51} C_VEL
LIN {X 0,Y 734.218,Z 826.182,A -85,B 0,C 180,E1 2149.378,E2 2149.378} C_VEL
LIN {X 0,Y 733.353,Z 875.743,A -85,B 0,C 180,E1 2151.17,E2 2151.17} C_VEL
LIN {X 0,Y 732.204,Z 920.756,A -85,B 0,C 180,E1 2153.334,E2 2153.334} C_VEL
LIN {X 0,Y 731.122,Z 965.282,A -85,B 0,C 180,E1 2156.074,E2 2156.074} C_VEL
LIN {X 0,Y 730.117,Z 1004.593,A -85,B 0,C 180,E1 2159.11,E2 2159.11} C_VEL
LIN {X 0,Y 729.402,Z 1038.848,A -85,B 0,C 180,E1 2162.374,E2 2162.374} C_VEL
LIN {X 0,Y 728.873,Z 1069.083,A -85,B 0,C 180,E1 2165.949,E2 2165.949} C_VEL
LIN {X 0,Y 728.566,Z 1093.064,A -85,B 0,C 180,E1 2169.55,E2 2169.55} C_VEL
LIN {X 0,Y 728.323,Z 1111.634,A -85,B 0,C 180,E1 2173.191,E2 2173.191} C_VEL
LIN {X 0,Y 728.266,Z 1125.196,A -85,B 0,C 180,E1 2176.886,E2 2176.886} C_VEL
LIN {X 0,Y 728.135,Z 1133.641,A -85,B 0,C 180,E1 2180.657,E2 2180.657} C_VEL
LIN {X 0,Y 728.074,Z 1136.892,A -85,B 0,C 180,E1 2184.523,E2 2184.523} C_VEL
LIN {X 0,Y 728.071,Z 1136.029,A -85,B 0,C 180,E1 2187.166,E2 2187.166} C_VEL
LIN {X 0,Y 728.284,Z 1130.87,A -85,B 0,C 180,E1 2190.771,E2 2190.771} C_VEL
LIN {X 0,Y 728.321,Z 1119.974,A -85,B 0,C 180,E1 2194.633,E2 2194.633} C_VEL
LIN {X 0,Y 728.405,Z 1103.296,A -85,B 0,C 180,E1 2198.485,E2 2198.485} C_VEL
LIN {X 0,Y 728.641,Z 1080.933,A -85,B 0,C 180,E1 2202.303,E2 2202.303} C_VEL
LIN {X 0,Y 729.074,Z 1053.295,A -85,B 0,C 180,E1 2205.925,E2 2205.925} C_VEL
LIN {X 0,Y 729.713,Z 1021.541,A -85,B 0,C 180,E1 2209.277,E2 2209.277} C_VEL
LIN {X 0,Y 730.676,Z 982.292,A -85,B 0,C 180,E1 2212.605,E2 2212.605} C_VEL
LIN {X 0,Y 731.716,Z 941.193,A -85,B 0,C 180,E1 2215.393,E2 2215.393} C_VEL
LIN {X 0,Y 732.898,Z 897.883,A -85,B 0,C 180,E1 2217.746,E2 2217.746} C_VEL
LIN {X 0,Y 733.854,Z 853.296,A -85,B 0,C 180,E1 2219.618,E2 2219.618} C_VEL
LIN {X 0,Y 733.775,Z 823.528,A -85,B 0,C 180,E1 2220.641,E2 2220.641} C_VEL
LIN {X 0,Y 727.736,Z 809.06,A -85,B 0,C 180,E1 2221.479,E2 2221.479} C_VEL
LIN {X 0,Y 727.623,Z 809.06,A -85,B 0,C 180,E1 2226.022,E2 2226.022} C_VEL
LIN {X 0,Y 727.77,Z 809.06,A -85,B 0,C 180,E1 2230.603,E2 2230.603} C_VEL
LIN {X 0,Y 727.89,Z 809.06,A -85,B 0,C 180,E1 2235.58,E2 2235.58} C_VEL
LIN {X 0,Y 728.082,Z 809.06,A -85,B 0,C 180,E1 2240.448,E2 2240.448} C_VEL
LIN {X 0,Y 727.976,Z 809.06,A -85,B 0,C 180,E1 2245.242,E2 2245.242} C_VEL
LIN {X 0,Y 728.008,Z 809.06,A -85,B 0,C 180,E1 2250.005,E2 2250.005} C_VEL
LIN {X 0,Y 728.121,Z 809.06,A -85,B 0,C 180,E1 2255.073,E2 2255.073} C_VEL
LIN {X 0,Y 728.009,Z 809.06,A -85,B 0,C 180,E1 2259.563,E2 2259.563} C_VEL
LIN {X 0,Y 727.92,Z 809.06,A -85,B 0,C 180,E1 2264.429,E2 2264.429} C_VEL
LIN {X 0,Y 727.963,Z 809.06,A -85,B 0,C 180,E1 2268.146,E2 2268.146} C_VEL
LIN {X 0,Y 727.918,Z 809.06,A -85,B 0,C 180,E1 2273.234,E2 2273.234} C_VEL
LIN {X 0,Y 727.906,Z 809.06,A -85,B 0,C 180,E1 2278.525,E2 2278.525} C_VEL
LIN {X 0,Y 727.919,Z 809.06,A -85,B 0,C 180,E1 2283.871,E2 2283.871} C_VEL
LIN {X 0,Y 727.702,Z 809.06,A -85,B 0,C 180,E1 2288.537,E2 2288.537} C_VEL
LIN {X 0,Y 728.007,Z 809.06,A -85,B 0,C 180,E1 2293.413,E2 2293.413} C_VEL
LIN {X 0,Y 727.671,Z 809.06,A -85,B 0,C 180,E1 2298.387,E2 2298.387} C_VEL
LIN {X 0,Y 727.681,Z 809.06,A -85,B 0,C 180,E1 2302.975,E2 2302.975} C_VEL
LIN {X 0,Y 727.714,Z 809.06,A -85,B 0,C 180,E1 2307.327,E2 2307.327} C_VEL
LIN {X 0,Y 727.84,Z 809.06,A -85,B 0,C 180,E1 2311.48,E2 2311.48} C_VEL
LIN {X 0,Y 727.879,Z 809.06,A -85,B 0,C 180,E1 2315.994,E2 2315.994} C_VEL
LIN {X 0,Y 727.951,Z 809.06,A -85,B 0,C 180,E1 2320.604,E2 2320.604} C_VEL
LIN {X 0,Y 727.964,Z 809.06,A -85,B 0,C 180,E1 2325.578,E2 2325.578} C_VEL
LIN {X 0,Y 728.063,Z 809.06,A -85,B 0,C 180,E1 2330.443,E2 2330.443} C_VEL
LIN {X 0,Y 727.976,Z 809.06,A -85,B 0,C 180,E1 2335.238,E2 2335.238} C_VEL
LIN {X 0,Y 728.108,Z 809.06,A -85,B 0,C 180,E1 2340,E2 2340} C_VEL
LIN {X 0,Y 728.18,Z 809.06,A -85,B 0,C 180,E1 2345.042,E2 2345.042} C_VEL
LIN {X 0,Y 728.012,Z 809.06,A -85,B 0,C 180,E1 2346.265,E2 2346.265} C_VEL
LIN {X 0,Y 724.073,Z 809.06,A -85,B 0,C 180,E1 2347.607,E2 2347.607} C_VEL
LIN {X 0,Y 720.139,Z 809.06,A -85,B 0,C 180,E1 2348.963,E2 2348.963} C_VEL
LIN {X 0,Y 720.082,Z 809.06,A -85,B 0,C 180,E1 2353.346,E2 2353.346} C_VEL
LIN {X 0,Y 720.007,Z 809.06,A -85,B 0,C 180,E1 2358.348,E2 2358.348} C_VEL
LIN {X 0,Y 720.007,Z 809.06,A -85,B 0,C 180,E1 2363.499,E2 2363.499} C_VEL
LIN {X 0,Y 719.952,Z 809.06,A -85,B 0,C 180,E1 2368.863,E2 2368.863} C_VEL
LIN {X 0,Y 720.014,Z 809.06,A -85,B 0,C 180,E1 2373.068,E2 2373.068} C_VEL
LIN {X 0,Y 719.933,Z 809.06,A -85,B 0,C 180,E1 2377.492,E2 2377.492} C_VEL
LIN {X 0,Y 720.032,Z 809.06,A -85,B 0,C 180,E1 2382.728,E2 2382.728} C_VEL
LIN {X 0,Y 719.757,Z 809.06,A -85,B 0,C 180,E1 2387.287,E2 2387.287} C_VEL
LIN {X 0,Y 720.124,Z 809.06,A -85,B 0,C 180,E1 2390.719,E2 2390.719} C_VEL
LIN {X 0,Y 724.417,Z 818.606,A -85,B 0,C 180,E1 2391.116,E2 2391.116} C_VEL
LIN {X 0,Y 729.13,Z 828.111,A -85,B 0,C 180,E1 2391.531,E2 2391.531} C_VEL
LIN {X 0,Y 728.966,Z 920.921,A -85,B 0,C 180,E1 2392.749,E2 2392.749} C_VEL
LIN {X 0,Y 727.98,Z 964.204,A -85,B 0,C 180,E1 2393.71,E2 2393.71} C_VEL
LIN {X 0,Y 726.91,Z 1012.825,A -85,B 0,C 180,E1 2395.326,E2 2395.326} C_VEL
LIN {X 0,Y 725.548,Z 1059.042,A -85,B 0,C 180,E1 2397.418,E2 2397.418} C_VEL
LIN {X 0,Y 724.385,Z 1101.185,A -85,B 0,C 180,E1 2399.857,E2 2399.857} C_VEL
LIN {X 0,Y 723.043,Z 1142.815,A -85,B 0,C 180,E1 2402.881,E2 2402.881} C_VEL
LIN {X 0,Y 722.021,Z 1177.865,A -85,B 0,C 180,E1 2406.034,E2 2406.034} C_VEL
LIN {X 0,Y 721.295,Z 1210.104,A -85,B 0,C 180,E1 2409.613,E2 2409.613} C_VEL
LIN {X 0,Y 720.855,Z 1235.89,A -85,B 0,C 180,E1 2413.243,E2 2413.243} C_VEL
LIN {X 0,Y 720.459,Z 1256.966,A -85,B 0,C 180,E1 2417.053,E2 2417.053} C_VEL
LIN {X 0,Y 720.325,Z 1272.338,A -85,B 0,C 180,E1 2420.943,E2 2420.943} C_VEL
LIN {X 0,Y 720.373,Z 1280.559,A -85,B 0,C 180,E1 2423.975,E2 2423.975} C_VEL
LIN {X 0,Y 720.253,Z 1285.87,A -85,B 0,C 180,E1 2427.59,E2 2427.59} C_VEL
LIN {X 0,Y 720.398,Z 1286.67,A -85,B 0,C 180,E1 2431.197,E2 2431.197} C_VEL
LIN {X 0,Y 720.191,Z 1282.919,A -85,B 0,C 180,E1 2434.809,E2 2434.809} C_VEL
LIN {X 0,Y 720.208,Z 1276.116,A -85,B 0,C 180,E1 2437.833,E2 2437.833} C_VEL
LIN {X 0,Y 720.395,Z 1263.416,A -85,B 0,C 180,E1 2441.489,E2 2441.489} C_VEL
LIN {X 0,Y 720.546,Z 1244.731,A -85,B 0,C 180,E1 2445.284,E2 2445.284} C_VEL
LIN {X 0,Y 720.904,Z 1223.585,A -85,B 0,C 180,E1 2448.597,E2 2448.597} C_VEL
LIN {X 0,Y 721.561,Z 1196.859,A -85,B 0,C 180,E1 2451.957,E2 2451.957} C_VEL
LIN {X 0,Y 722.482,Z 1161.875,A -85,B 0,C 180,E1 2455.489,E2 2455.489} C_VEL
LIN {X 0,Y 723.572,Z 1123.916,A -85,B 0,C 180,E1 2458.573,E2 2458.573} C_VEL
LIN {X 0,Y 724.916,Z 1081.872,A -85,B 0,C 180,E1 2461.333,E2 2461.333} C_VEL
LIN {X 0,Y 726.281,Z 1036.983,A -85,B 0,C 180,E1 2463.646,E2 2463.646} C_VEL
LIN {X 0,Y 727.543,Z 992.206,A -85,B 0,C 180,E1 2465.423,E2 2465.423} C_VEL
LIN {X 0,Y 728.449,Z 946.127,A -85,B 0,C 180,E1 2466.742,E2 2466.742} C_VEL
LIN {X 0,Y 729.121,Z 901.155,A -85,B 0,C 180,E1 2467.564,E2 2467.564} C_VEL
LIN {X 0,Y 728.375,Z 825.992,A -85,B 0,C 180,E1 2468.542,E2 2468.542} C_VEL
LIN {X 0,Y 719.807,Z 809.452,A -85,B 0,C 180,E1 2469.296,E2 2469.296} C_VEL
LIN {X 0,Y 720.082,Z 809.06,A -85,B 0,C 180,E1 2474.484,E2 2474.484} C_VEL
LIN {X 0,Y 719.876,Z 809.06,A -85,B 0,C 180,E1 2479.407,E2 2479.407} C_VEL
LIN {X 0,Y 719.851,Z 809.06,A -85,B 0,C 180,E1 2484.004,E2 2484.004} C_VEL
LIN {X 0,Y 719.859,Z 809.06,A -85,B 0,C 180,E1 2489.377,E2 2489.377} C_VEL
LIN {X 0,Y 719.858,Z 809.06,A -85,B 0,C 180,E1 2494.492,E2 2494.492} C_VEL
LIN {X 0,Y 719.896,Z 809.06,A -85,B 0,C 180,E1 2500.377,E2 2500.377} C_VEL
LIN {X 0,Y 719.914,Z 809.06,A -85,B 0,C 180,E1 2505.412,E2 2505.412} C_VEL
LIN {X 0,Y 719.791,Z 809.06,A -85,B 0,C 180,E1 2508.034,E2 2508.034} C_VEL
LIN {X 0,Y 727.614,Z 829.235,A -85,B 0,C 180,E1 2509.107,E2 2509.107} C_VEL
LIN {X 0,Y 726.57,Z 877.266,A -85,B 0,C 180,E1 2510.876,E2 2510.876} C_VEL
LIN {X 0,Y 725.192,Z 921.651,A -85,B 0,C 180,E1 2513.044,E2 2513.044} C_VEL
LIN {X 0,Y 723.895,Z 964.95,A -85,B 0,C 180,E1 2515.735,E2 2515.735} C_VEL
LIN {X 0,Y 722.688,Z 1004.332,A -85,B 0,C 180,E1 2518.802,E2 2518.802} C_VEL
LIN {X 0,Y 721.763,Z 1038.646,A -85,B 0,C 180,E1 2522.099,E2 2522.099} C_VEL
LIN {X 0,Y 721.143,Z 1069.708,A -85,B 0,C 180,E1 2525.819,E2 2525.819} C_VEL
LIN {X 0,Y 720.712,Z 1094.632,A -85,B 0,C 180,E1 2529.655,E2 2529.655} C_VEL
LIN {X 0,Y 720.399,Z 1112.864,A -85,B 0,C 180,E1 2533.339,E2 2533.339} C_VEL
LIN {X 0,Y 720.343,Z 1125.992,A -85,B 0,C 180,E1 2537.077,E2 2537.077} C_VEL
LIN {X 0,Y 720.223,Z 1134.086,A -85,B 0,C 180,E1 2540.894,E2 2540.894} C_VEL
LIN {X 0,Y 720.131,Z 1136.972,A -85,B 0,C 180,E1 2544.812,E2 2544.812} C_VEL
LIN {X 0,Y 720.158,Z 1134.311,A -85,B 0,C 180,E1 2548.853,E2 2548.853} C_VEL
LIN {X 0,Y 720.223,Z 1127.947,A -85,B 0,C 180,E1 2552.105,E2 2552.105} C_VEL
LIN {X 0,Y 720.28,Z 1117.036,A -85,B 0,C 180,E1 2555.521,E2 2555.521} C_VEL
LIN {X 0,Y 720.495,Z 1100.903,A -85,B 0,C 180,E1 2559.114,E2 2559.114} C_VEL
LIN {X 0,Y 720.771,Z 1079.958,A -85,B 0,C 180,E1 2562.64,E2 2562.64} C_VEL
LIN {X 0,Y 721.392,Z 1052.296,A -85,B 0,C 180,E1 2566.28,E2 2566.28} C_VEL
LIN {X 0,Y 722.184,Z 1021.311,A -85,B 0,C 180,E1 2569.569,E2 2569.569} C_VEL
LIN {X 0,Y 723.326,Z 982.575,A -85,B 0,C 180,E1 2572.888,E2 2572.888} C_VEL
LIN {X 0,Y 724.575,Z 942.826,A -85,B 0,C 180,E1 2575.622,E2 2575.622} C_VEL
LIN {X 0,Y 725.978,Z 899.641,A -85,B 0,C 180,E1 2578.009,E2 2578.009} C_VEL
LIN {X 0,Y 727.146,Z 855.924,A -85,B 0,C 180,E1 2579.885,E2 2579.885} C_VEL
LIN {X 0,Y 727.232,Z 826.982,A -85,B 0,C 180,E1 2580.902,E2 2580.902} C_VEL
LIN {X 0,Y 719.842,Z 809.06,A -85,B 0,C 180,E1 2581.887,E2 2581.887} C_VEL
LIN {X 0,Y 719.669,Z 809.06,A -85,B 0,C 180,E1 2586.494,E2 2586.494} C_VEL
LIN {X 0,Y 719.815,Z 809.06,A -85,B 0,C 180,E1 2590.839,E2 2590.839} C_VEL
LIN {X 0,Y 719.963,Z 809.06,A -85,B 0,C 180,E1 2596.657,E2 2596.657} C_VEL
LIN {X 0,Y 720.184,Z 809.06,A -85,B 0,C 180,E1 2600.429,E2 2600.429} C_VEL
LIN {X 0,Y 720.095,Z 809.06,A -85,B 0,C 180,E1 2605.19,E2 2605.19} C_VEL
LIN {X 0,Y 720.126,Z 809.06,A -85,B 0,C 180,E1 2610.005,E2 2610.005} C_VEL
LIN {X 0,Y 720.302,Z 809.06,A -85,B 0,C 180,E1 2614.818,E2 2614.818} C_VEL
LIN {X 0,Y 720.111,Z 809.06,A -85,B 0,C 180,E1 2619.669,E2 2619.669} C_VEL
LIN {X 0,Y 720.018,Z 809.06,A -85,B 0,C 180,E1 2624.591,E2 2624.591} C_VEL
LIN {X 0,Y 720.086,Z 809.06,A -85,B 0,C 180,E1 2629.223,E2 2629.223} C_VEL
LIN {X 0,Y 719.98,Z 809.06,A -85,B 0,C 180,E1 2634.824,E2 2634.824} C_VEL
LIN {X 0,Y 719.913,Z 809.06,A -85,B 0,C 180,E1 2640.254,E2 2640.254} C_VEL
LIN {X 0,Y 719.904,Z 809.06,A -85,B 0,C 180,E1 2644.528,E2 2644.528} C_VEL
LIN {X 0,Y 719.749,Z 809.06,A -85,B 0,C 180,E1 2649.043,E2 2649.043} C_VEL
LIN {X 0,Y 720.065,Z 809.06,A -85,B 0,C 180,E1 2654.484,E2 2654.484} C_VEL
LIN {X 0,Y 719.848,Z 809.06,A -85,B 0,C 180,E1 2659.406,E2 2659.406} C_VEL
LIN {X 0,Y 719.823,Z 809.06,A -85,B 0,C 180,E1 2664.962,E2 2664.962} C_VEL
LIN {X 0,Y 719.946,Z 809.06,A -85,B 0,C 180,E1 2669.755,E2 2669.755} C_VEL
LIN {X 0,Y 720.089,Z 809.06,A -85,B 0,C 180,E1 2674.476,E2 2674.476} C_VEL
LIN {X 0,Y 720.033,Z 809.06,A -85,B 0,C 180,E1 2679.1,E2 2679.1} C_VEL
LIN {X 0,Y 720.089,Z 809.06,A -85,B 0,C 180,E1 2684.171,E2 2684.171} C_VEL
LIN {X 0,Y 720.22,Z 809.06,A -85,B 0,C 180,E1 2689.117,E2 2689.117} C_VEL
LIN {X 0,Y 720.197,Z 809.06,A -85,B 0,C 180,E1 2693.979,E2 2693.979} C_VEL
LIN {X 0,Y 720.109,Z 809.06,A -85,B 0,C 180,E1 2698.798,E2 2698.798} C_VEL
LIN {X 0,Y 720.13,Z 809.06,A -85,B 0,C 180,E1 2702.406,E2 2702.406} C_VEL
LIN {X 0,Y 720.112,Z 809.06,A -85,B 0,C 180,E1 2706.26,E2 2706.26} C_VEL
LIN {X 0,Y 720.139,Z 809.06,A -85,B 0,C 180,E1 2708.963,E2 2708.963} C_VEL
LIN {X 0,Y 716.102,Z 809.06,A -85,B 0,C 180,E1 2710.318,E2 2710.318} C_VEL
LIN {X 0,Y 712.15,Z 809.06,A -85,B 0,C 180,E1 2711.688,E2 2711.688} C_VEL
LIN {X 0,Y 712.232,Z 809.06,A -85,B 0,C 180,E1 2717.294,E2 2717.294} C_VEL
LIN {X 0,Y 712.032,Z 809.06,A -85,B 0,C 180,E1 2722.457,E2 2722.457} C_VEL
LIN {X 0,Y 711.964,Z 809.06,A -85,B 0,C 180,E1 2726.94,E2 2726.94} C_VEL
LIN {X 0,Y 712.053,Z 809.06,A -85,B 0,C 180,E1 2732.04,E2 2732.04} C_VEL
LIN {X 0,Y 712.029,Z 809.06,A -85,B 0,C 180,E1 2736.455,E2 2736.455} C_VEL
LIN {X 0,Y 712.069,Z 809.06,A -85,B 0,C 180,E1 2742.029,E2 2742.029} C_VEL
LIN {X 0,Y 711.971,Z 809.06,A -85,B 0,C 180,E1 2746.185,E2 2746.185} C_VEL
LIN {X 0,Y 712.202,Z 809.497,A -85,B 0,C 180,E1 2750.202,E2 2750.202} C_VEL
LIN {X 0,Y 722.787,Z 829.833,A -85,B 0,C 180,E1 2751.152,E2 2751.152} C_VEL
LIN {X 0,Y 722.639,Z 921.799,A -85,B 0,C 180,E1 2752.384,E2 2752.384} C_VEL
LIN {X 0,Y 721.508,Z 965.755,A -85,B 0,C 180,E1 2753.377,E2 2753.377} C_VEL
LIN {X 0,Y 720.259,Z 1013.45,A -85,B 0,C 180,E1 2754.986,E2 2754.986} C_VEL
LIN {X 0,Y 718.61,Z 1060.861,A -85,B 0,C 180,E1 2757.161,E2 2757.161} C_VEL
LIN {X 0,Y 717.17,Z 1102.572,A -85,B 0,C 180,E1 2759.619,E2 2759.619} C_VEL
LIN {X 0,Y 715.604,Z 1145.093,A -85,B 0,C 180,E1 2762.761,E2 2762.761} C_VEL
LIN {X 0,Y 714.396,Z 1180.89,A -85,B 0,C 180,E1 2766.073,E2 2766.073} C_VEL
LIN {X 0,Y 713.538,Z 1211.33,A -85,B 0,C 180,E1 2769.543,E2 2769.543} C_VEL
LIN {X 0,Y 712.994,Z 1237.866,A -85,B 0,C 180,E1 2773.37,E2 2773.37} C_VEL
LIN {X 0,Y 712.601,Z 1257.176,A -85,B 0,C 180,E1 2776.95,E2 2776.95} C_VEL
LIN {X 0,Y 712.457,Z 1272.533,A -85,B 0,C 180,E1 2780.904,E2 2780.904} C_VEL
LIN {X 0,Y 712.402,Z 1281.789,A -85,B 0,C 180,E1 2784.518,E2 2784.518} C_VEL
LIN {X 0,Y 712.35,Z 1285.87,A -85,B 0,C 180,E1 2787.564,E2 2787.564} C_VEL
LIN {X 0,Y 712.496,Z 1286.67,A -85,B 0,C 180,E1 2791.21,E2 2791.21} C_VEL
LIN {X 0,Y 712.299,Z 1282.919,A -85,B 0,C 180,E1 2794.863,E2 2794.863} C_VEL
LIN {X 0,Y 712.306,Z 1276.116,A -85,B 0,C 180,E1 2797.921,E2 2797.921} C_VEL
LIN {X 0,Y 712.516,Z 1263.415,A -85,B 0,C 180,E1 2801.618,E2 2801.618} C_VEL
LIN {X 0,Y 712.724,Z 1244.733,A -85,B 0,C 180,E1 2805.456,E2 2805.456} C_VEL
LIN {X 0,Y 713.151,Z 1223.759,A -85,B 0,C 180,E1 2808.782,E2 2808.782} C_VEL
LIN {X 0,Y 713.917,Z 1196.509,A -85,B 0,C 180,E1 2812.244,E2 2812.244} C_VEL
LIN {X 0,Y 715.02,Z 1161.262,A -85,B 0,C 180,E1 2815.833,E2 2815.833} C_VEL
LIN {X 0,Y 716.291,Z 1123.917,A -85,B 0,C 180,E1 2818.891,E2 2818.891} C_VEL
LIN {X 0,Y 717.874,Z 1082.73,A -85,B 0,C 180,E1 2821.626,E2 2821.626} C_VEL
LIN {X 0,Y 719.466,Z 1038.425,A -85,B 0,C 180,E1 2823.938,E2 2823.938} C_VEL
LIN {X 0,Y 720.916,Z 994.267,A -85,B 0,C 180,E1 2825.72,E2 2825.72} C_VEL
LIN {X 0,Y 721.989,Z 948.901,A -85,B 0,C 180,E1 2827.055,E2 2827.055} C_VEL
LIN {X 0,Y 722.795,Z 903.356,A -85,B 0,C 180,E1 2827.918,E2 2827.918} C_VEL
LIN {X 0,Y 722.341,Z 829.418,A -85,B 0,C 180,E1 2828.882,E2 2828.882} C_VEL
LIN {X 0,Y 711.891,Z 809.694,A -85,B 0,C 180,E1 2829.817,E2 2829.817} C_VEL
LIN {X 0,Y 712.181,Z 809.06,A -85,B 0,C 180,E1 2834.433,E2 2834.433} C_VEL
LIN {X 0,Y 711.937,Z 809.06,A -85,B 0,C 180,E1 2839.817,E2 2839.817} C_VEL
LIN {X 0,Y 711.957,Z 809.06,A -85,B 0,C 180,E1 2845.038,E2 2845.038} C_VEL
LIN {X 0,Y 711.885,Z 809.06,A -85,B 0,C 180,E1 2850.479,E2 2850.479} C_VEL
LIN {X 0,Y 711.929,Z 809.06,A -85,B 0,C 180,E1 2854.882,E2 2854.882} C_VEL
LIN {X 0,Y 711.967,Z 809.06,A -85,B 0,C 180,E1 2860.149,E2 2860.149} C_VEL
LIN {X 0,Y 711.998,Z 809.06,A -85,B 0,C 180,E1 2865.246,E2 2865.246} C_VEL
LIN {X 0,Y 711.894,Z 809.375,A -85,B 0,C 180,E1 2867.567,E2 2867.567} C_VEL
LIN {X 0,Y 720.985,Z 833.051,A -85,B 0,C 180,E1 2868.853,E2 2868.853} C_VEL
LIN {X 0,Y 719.762,Z 880.112,A -85,B 0,C 180,E1 2870.636,E2 2870.636} C_VEL
LIN {X 0,Y 718.062,Z 925.229,A -85,B 0,C 180,E1 2872.898,E2 2872.898} C_VEL
LIN {X 0,Y 716.642,Z 967.801,A -85,B 0,C 180,E1 2875.616,E2 2875.616} C_VEL
LIN {X 0,Y 715.163,Z 1007.562,A -85,B 0,C 180,E1 2878.789,E2 2878.789} C_VEL
LIN {X 0,Y 714.102,Z 1041.171,A -85,B 0,C 180,E1 2882.122,E2 2882.122} C_VEL
LIN {X 0,Y 713.372,Z 1070.999,A -85,B 0,C 180,E1 2885.779,E2 2885.779} C_VEL
LIN {X 0,Y 712.863,Z 1096.199,A -85,B 0,C 180,E1 2889.762,E2 2889.762} C_VEL
LIN {X 0,Y 712.521,Z 1114.074,A -85,B 0,C 180,E1 2893.489,E2 2893.489} C_VEL
LIN {X 0,Y 712.398,Z 1127.027,A -85,B 0,C 180,E1 2897.371,E2 2897.371} C_VEL
LIN {X 0,Y 712.274,Z 1134.47,A -85,B 0,C 180,E1 2901.138,E2 2901.138} C_VEL
LIN {X 0,Y 712.218,Z 1136.971,A -85,B 0,C 180,E1 2905.106,E2 2905.106} C_VEL
LIN {X 0,Y 712.258,Z 1133.866,A -85,B 0,C 180,E1 2909.204,E2 2909.204} C_VEL
LIN {X 0,Y 712.35,Z 1126.674,A -85,B 0,C 180,E1 2912.67,E2 2912.67} C_VEL
LIN {X 0,Y 712.388,Z 1114.551,A -85,B 0,C 180,E1 2916.3,E2 2916.3} C_VEL
LIN {X 0,Y 712.636,Z 1099.09,A -85,B 0,C 180,E1 2919.63,E2 2919.63} C_VEL
LIN {X 0,Y 713.064,Z 1077.373,A -85,B 0,C 180,E1 2923.213,E2 2923.213} C_VEL
LIN {X 0,Y 713.751,Z 1050.343,A -85,B 0,C 180,E1 2926.757,E2 2926.757} C_VEL
LIN {X 0,Y 714.699,Z 1019.419,A -85,B 0,C 180,E1 2930.024,E2 2930.024} C_VEL
LIN {X 0,Y 716.086,Z 981.201,A -85,B 0,C 180,E1 2933.304,E2 2933.304} C_VEL
LIN {X 0,Y 717.654,Z 939.495,A -85,B 0,C 180,E1 2936.164,E2 2936.164} C_VEL
LIN {X 0,Y 719.213,Z 896.891,A -85,B 0,C 180,E1 2938.5,E2 2938.5} C_VEL
LIN {X 0,Y 720.603,Z 853.268,A -85,B 0,C 180,E1 2940.352,E2 2940.352} C_VEL
LIN {X 0,Y 720.658,Z 830.238,A -85,B 0,C 180,E1 2941.173,E2 2941.173} C_VEL
LIN {X 0,Y 711.97,Z 809.06,A -85,B 0,C 180,E1 2942.404,E2 2942.404} C_VEL
LIN {X 0,Y 711.759,Z 809.06,A -85,B 0,C 180,E1 2947.539,E2 2947.539} C_VEL
LIN {X 0,Y 711.786,Z 809.06,A -85,B 0,C 180,E1 2951.437,E2 2951.437} C_VEL
LIN {X 0,Y 712.065,Z 809.06,A -85,B 0,C 180,E1 2956.506,E2 2956.506} C_VEL
LIN {X 0,Y 712.289,Z 809.06,A -85,B 0,C 180,E1 2960.234,E2 2960.234} C_VEL
LIN {X 0,Y 712.212,Z 809.06,A -85,B 0,C 180,E1 2965.137,E2 2965.137} C_VEL
LIN {X 0,Y 712.226,Z 809.06,A -85,B 0,C 180,E1 2970.005,E2 2970.005} C_VEL
LIN {X 0,Y 712.391,Z 809.06,A -85,B 0,C 180,E1 2974.872,E2 2974.872} C_VEL
LIN {X 0,Y 712.192,Z 809.06,A -85,B 0,C 180,E1 2979.777,E2 2979.777} C_VEL
LIN {X 0,Y 712.138,Z 809.06,A -85,B 0,C 180,E1 2984.756,E2 2984.756} C_VEL
LIN {X 0,Y 712.162,Z 809.06,A -85,B 0,C 180,E1 2988.563,E2 2988.563} C_VEL
LIN {X 0,Y 712.086,Z 809.06,A -85,B 0,C 180,E1 2993.782,E2 2993.782} C_VEL
LIN {X 0,Y 712.023,Z 809.06,A -85,B 0,C 180,E1 2999.222,E2 2999.222} C_VEL
LIN {X 0,Y 712.029,Z 809.06,A -85,B 0,C 180,E1 3004.146,E2 3004.146} C_VEL
LIN {X 0,Y 711.878,Z 809.06,A -85,B 0,C 180,E1 3008.249,E2 3008.249} C_VEL
LIN {X 0,Y 712.161,Z 809.06,A -85,B 0,C 180,E1 3013.832,E2 3013.832} C_VEL
LIN {X 0,Y 711.857,Z 809.06,A -85,B 0,C 180,E1 3018.853,E2 3018.853} C_VEL
LIN {X 0,Y 711.922,Z 809.06,A -85,B 0,C 180,E1 3023.768,E2 3023.768} C_VEL
LIN {X 0,Y 712.007,Z 809.06,A -85,B 0,C 180,E1 3029.382,E2 3029.382} C_VEL
LIN {X 0,Y 712.187,Z 809.06,A -85,B 0,C 180,E1 3033.543,E2 3033.543} C_VEL
LIN {X 0,Y 712.125,Z 809.06,A -85,B 0,C 180,E1 3039.021,E2 3039.021} C_VEL
LIN {X 0,Y 712.174,Z 809.06,A -85,B 0,C 180,E1 3043.99,E2 3043.99} C_VEL
LIN {X 0,Y 712.276,Z 809.06,A -85,B 0,C 180,E1 3048.994,E2 3048.994} C_VEL
LIN {X 0,Y 712.317,Z 809.06,A -85,B 0,C 180,E1 3053.912,E2 3053.912} C_VEL
LIN {X 0,Y 712.21,Z 809.06,A -85,B 0,C 180,E1 3058.785,E2 3058.785} C_VEL
LIN {X 0,Y 712.229,Z 809.06,A -85,B 0,C 180,E1 3062.432,E2 3062.432} C_VEL
LIN {X 0,Y 712.234,Z 809.06,A -85,B 0,C 180,E1 3066.09,E2 3066.09} C_VEL
LIN {X 0,Y 712.16,Z 809.06,A -85,B 0,C 180,E1 3071.009,E2 3071.009} C_VEL
LIN {X 0,Y 712.15,Z 809.06,A -85,B 0,C 180,E1 3071.688,E2 3071.688} C_VEL
LIN {X 0,Y 710.914,Z 809.06,A -85,B 0,C 180,E1 3072.384,E2 3072.384} C_VEL
LIN {X 0,Y 704.289,Z 809.06,A -85,B 0,C 180,E1 3074.271,E2 3074.271} C_VEL
LIN {X 0,Y 704.199,Z 809.06,A -85,B 0,C 180,E1 3074.45,E2 3074.45} C_VEL
LIN {X 0,Y 704.2,Z 809.06,A -85,B 0,C 180,E1 3079.227,E2 3079.227} C_VEL
LIN {X 0,Y 704.181,Z 809.06,A -85,B 0,C 180,E1 3084.06,E2 3084.06} C_VEL
LIN {X 0,Y 704.085,Z 809.06,A -85,B 0,C 180,E1 3089.577,E2 3089.577} C_VEL
LIN {X 0,Y 704.085,Z 809.06,A -85,B 0,C 180,E1 3093.916,E2 3093.916} C_VEL
LIN {X 0,Y 703.965,Z 809.06,A -85,B 0,C 180,E1 3098.496,E2 3098.496} C_VEL
LIN {X 0,Y 704.249,Z 809.06,A -85,B 0,C 180,E1 3103.36,E2 3103.36} C_VEL
LIN {X 0,Y 703.997,Z 809.06,A -85,B 0,C 180,E1 3108.696,E2 3108.696} C_VEL
LIN {X 0,Y 704.149,Z 809.251,A -85,B 0,C 180,E1 3109.65,E2 3109.65} C_VEL
LIN {X 0,Y 706.691,Z 814.815,A -85,B 0,C 180,E1 3109.898,E2 3109.898} C_VEL
LIN {X 0,Y 716.896,Z 834.961,A -85,B 0,C 180,E1 3110.836,E2 3110.836} C_VEL
LIN {X 0,Y 716.399,Z 920.092,A -85,B 0,C 180,E1 3111.966,E2 3111.966} C_VEL
LIN {X 0,Y 715.153,Z 964.086,A -85,B 0,C 180,E1 3112.95,E2 3112.95} C_VEL
LIN {X 0,Y 713.663,Z 1012.292,A -85,B 0,C 180,E1 3114.564,E2 3114.564} C_VEL
LIN {X 0,Y 711.826,Z 1059.042,A -85,B 0,C 180,E1 3116.709,E2 3116.709} C_VEL
LIN {X 0,Y 710.091,Z 1100.684,A -85,B 0,C 180,E1 3119.151,E2 3119.151} C_VEL
LIN {X 0,Y 708.304,Z 1143.086,A -85,B 0,C 180,E1 3122.291,E2 3122.291} C_VEL
LIN {X 0,Y 706.939,Z 1177.359,A -85,B 0,C 180,E1 3125.436,E2 3125.436} C_VEL
LIN {X 0,Y 705.926,Z 1210.104,A -85,B 0,C 180,E1 3129.148,E2 3129.148} C_VEL
LIN {X 0,Y 705.213,Z 1235.894,A -85,B 0,C 180,E1 3132.86,E2 3132.86} C_VEL
LIN {X 0,Y 704.769,Z 1256.909,A -85,B 0,C 180,E1 3136.748,E2 3136.748} C_VEL
LIN {X 0,Y 704.585,Z 1271.808,A -85,B 0,C 180,E1 3140.568,E2 3140.568} C_VEL
LIN {X 0,Y 704.514,Z 1281.789,A -85,B 0,C 180,E1 3144.456,E2 3144.456} C_VEL
LIN {X 0,Y 704.465,Z 1285.871,A -85,B 0,C 180,E1 3147.536,E2 3147.536} C_VEL
LIN {X 0,Y 704.594,Z 1286.67,A -85,B 0,C 180,E1 3151.224,E2 3151.224} C_VEL
LIN {X 0,Y 704.399,Z 1282.919,A -85,B 0,C 180,E1 3154.917,E2 3154.917} C_VEL
LIN {X 0,Y 704.4,Z 1276.116,A -85,B 0,C 180,E1 3158.01,E2 3158.01} C_VEL
LIN {X 0,Y 704.643,Z 1263.414,A -85,B 0,C 180,E1 3161.749,E2 3161.749} C_VEL
LIN {X 0,Y 704.863,Z 1246.02,A -85,B 0,C 180,E1 3165.4,E2 3165.4} C_VEL
LIN {X 0,Y 705.364,Z 1224.146,A -85,B 0,C 180,E1 3168.94,E2 3168.94} C_VEL
LIN {X 0,Y 706.246,Z 1196.67,A -85,B 0,C 180,E1 3172.48,E2 3172.48} C_VEL
LIN {X 0,Y 707.563,Z 1161.32,A -85,B 0,C 180,E1 3176.12,E2 3176.12} C_VEL
LIN {X 0,Y 709.122,Z 1123.816,A -85,B 0,C 180,E1 3179.219,E2 3179.219} C_VEL
LIN {X 0,Y 710.884,Z 1082.983,A -85,B 0,C 180,E1 3181.958,E2 3181.958} C_VEL
LIN {X 0,Y 712.676,Z 1039.319,A -85,B 0,C 180,E1 3184.263,E2 3184.263} C_VEL
LIN {X 0,Y 714.312,Z 995.891,A -85,B 0,C 180,E1 3186.039,E2 3186.039} C_VEL
LIN {X 0,Y 715.604,Z 950.213,A -85,B 0,C 180,E1 3187.409,E2 3187.409} C_VEL
LIN {X 0,Y 716.55,Z 903.684,A -85,B 0,C 180,E1 3188.302,E2 3188.302} C_VEL
LIN {X 0,Y 716.234,Z 832.833,A -85,B 0,C 180,E1 3189.234,E2 3189.234} C_VEL
LIN {X 0,Y 704.099,Z 810.566,A -85,B 0,C 180,E1 3190.336,E2 3190.336} C_VEL
LIN {X 0,Y 703.979,Z 809.06,A -85,B 0,C 180,E1 3190.391,E2 3190.391} C_VEL
LIN {X 0,Y 704.208,Z 809.06,A -85,B 0,C 180,E1 3195.073,E2 3195.073} C_VEL
LIN {X 0,Y 704.05,Z 809.06,A -85,B 0,C 180,E1 3200.583,E2 3200.583} C_VEL
LIN {X 0,Y 703.977,Z 809.06,A -85,B 0,C 180,E1 3206.078,E2 3206.078} C_VEL
LIN {X 0,Y 703.998,Z 809.06,A -85,B 0,C 180,E1 3210.419,E2 3210.419} C_VEL
LIN {X 0,Y 704.005,Z 809.06,A -85,B 0,C 180,E1 3214.579,E2 3214.579} C_VEL
LIN {X 0,Y 704.063,Z 809.06,A -85,B 0,C 180,E1 3219.917,E2 3219.917} C_VEL
LIN {X 0,Y 704.052,Z 809.06,A -85,B 0,C 180,E1 3225.076,E2 3225.076} C_VEL
LIN {X 0,Y 704.025,Z 809.145,A -85,B 0,C 180,E1 3227.069,E2 3227.069} C_VEL
LIN {X 0,Y 714.458,Z 834.756,A -85,B 0,C 180,E1 3228.528,E2 3228.528} C_VEL
LIN {X 0,Y 713.016,Z 881.204,A -85,B 0,C 180,E1 3230.316,E2 3230.316} C_VEL
LIN {X 0,Y 711.079,Z 926.167,A -85,B 0,C 180,E1 3232.6,E2 3232.6} C_VEL
LIN {X 0,Y 709.354,Z 968.542,A -85,B 0,C 180,E1 3235.341,E2 3235.341} C_VEL
LIN {X 0,Y 707.668,Z 1009.017,A -85,B 0,C 180,E1 3238.623,E2 3238.623} C_VEL
LIN {X 0,Y 706.427,Z 1043.7,A -85,B 0,C 180,E1 3242.145,E2 3242.145} C_VEL
LIN {X 0,Y 705.607,Z 1071.922,A -85,B 0,C 180,E1 3245.692,E2 3245.692} C_VEL
LIN {X 0,Y 705.039,Z 1096.656,A -85,B 0,C 180,E1 3249.672,E2 3249.672} C_VEL
LIN {X 0,Y 704.664,Z 1113.708,A -85,B 0,C 180,E1 3253.272,E2 3253.272} C_VEL
LIN {X 0,Y 704.545,Z 1125.806,A -85,B 0,C 180,E1 3256.829,E2 3256.829} C_VEL
LIN {X 0,Y 704.443,Z 1132.961,A -85,B 0,C 180,E1 3260.071,E2 3260.071} C_VEL
LIN {X 0,Y 704.293,Z 1136.772,A -85,B 0,C 180,E1 3264.055,E2 3264.055} C_VEL
LIN {X 0,Y 704.294,Z 1135.255,A -85,B 0,C 180,E1 3268.163,E2 3268.163} C_VEL
LIN {X 0,Y 704.514,Z 1129.427,A -85,B 0,C 180,E1 3271.645,E2 3271.645} C_VEL
LIN {X 0,Y 704.541,Z 1118.29,A -85,B 0,C 180,E1 3275.422,E2 3275.422} C_VEL
LIN {X 0,Y 704.775,Z 1102.213,A -85,B 0,C 180,E1 3279.17,E2 3279.17} C_VEL
LIN {X 0,Y 705.172,Z 1082.119,A -85,B 0,C 180,E1 3282.71,E2 3282.71} C_VEL
LIN {X 0,Y 705.943,Z 1056.432,A -85,B 0,C 180,E1 3286.263,E2 3286.263} C_VEL
LIN {X 0,Y 707.04,Z 1024.029,A -85,B 0,C 180,E1 3289.862,E2 3289.862} C_VEL
LIN {X 0,Y 708.575,Z 986.255,A -85,B 0,C 180,E1 3293.22,E2 3293.22} C_VEL
LIN {X 0,Y 710.298,Z 946.65,A -85,B 0,C 180,E1 3296.06,E2 3296.06} C_VEL
LIN {X 0,Y 712.193,Z 902.332,A -85,B 0,C 180,E1 3298.592,E2 3298.592} C_VEL
LIN {X 0,Y 713.84,Z 858.968,A -85,B 0,C 180,E1 3300.515,E2 3300.515} C_VEL
LIN {X 0,Y 713.932,Z 832.843,A -85,B 0,C 180,E1 3301.481,E2 3301.481} C_VEL
LIN {X 0,Y 704.058,Z 809.06,A -85,B 0,C 180,E1 3302.844,E2 3302.844} C_VEL
LIN {X 0,Y 703.953,Z 809.06,A -85,B 0,C 180,E1 3308.604,E2 3308.604} C_VEL
LIN {X 0,Y 703.874,Z 809.06,A -85,B 0,C 180,E1 3313.8,E2 3313.8} C_VEL
LIN {X 0,Y 704.34,Z 809.06,A -85,B 0,C 180,E1 3318.873,E2 3318.873} C_VEL
LIN {X 0,Y 704.372,Z 809.06,A -85,B 0,C 180,E1 3323.848,E2 3323.848} C_VEL
LIN {X 0,Y 704.272,Z 809.06,A -85,B 0,C 180,E1 3328.776,E2 3328.776} C_VEL
LIN {X 0,Y 704.274,Z 809.06,A -85,B 0,C 180,E1 3332.464,E2 3332.464} C_VEL
LIN {X 0,Y 704.288,Z 809.06,A -85,B 0,C 180,E1 3336.163,E2 3336.163} C_VEL
LIN {X 0,Y 704.236,Z 809.06,A -85,B 0,C 180,E1 3341.139,E2 3341.139} C_VEL
LIN {X 0,Y 704.312,Z 809.06,A -85,B 0,C 180,E1 3346.2,E2 3346.2} C_VEL
LIN {X 0,Y 704.178,Z 809.06,A -85,B 0,C 180,E1 3351.4,E2 3351.4} C_VEL
LIN {X 0,Y 704.098,Z 809.06,A -85,B 0,C 180,E1 3355.67,E2 3355.67} C_VEL
LIN {X 0,Y 704.098,Z 809.06,A -85,B 0,C 180,E1 3361.007,E2 3361.007} C_VEL
LIN {X 0,Y 704.067,Z 809.06,A -85,B 0,C 180,E1 3365.419,E2 3365.419} C_VEL
LIN {X 0,Y 703.886,Z 809.06,A -85,B 0,C 180,E1 3370.098,E2 3370.098} C_VEL
LIN {X 0,Y 704.193,Z 809.06,A -85,B 0,C 180,E1 3375.088,E2 3375.088} C_VEL
LIN {X 0,Y 704.033,Z 809.06,A -85,B 0,C 180,E1 3380.601,E2 3380.601} C_VEL
LIN {X 0,Y 703.983,Z 809.06,A -85,B 0,C 180,E1 3386.08,E2 3386.08} C_VEL
LIN {X 0,Y 704.099,Z 809.06,A -85,B 0,C 180,E1 3390.425,E2 3390.425} C_VEL
LIN {X 0,Y 704.215,Z 809.06,A -85,B 0,C 180,E1 3394.588,E2 3394.588} C_VEL
LIN {X 0,Y 704.206,Z 809.06,A -85,B 0,C 180,E1 3399.922,E2 3399.922} C_VEL
LIN {X 0,Y 704.243,Z 809.06,A -85,B 0,C 180,E1 3405.081,E2 3405.081} C_VEL
LIN {X 0,Y 704.377,Z 809.06,A -85,B 0,C 180,E1 3410.119,E2 3410.119} C_VEL
LIN {X 0,Y 704.312,Z 809.06,A -85,B 0,C 180,E1 3415.078,E2 3415.078} C_VEL
LIN {X 0,Y 704.425,Z 809.06,A -85,B 0,C 180,E1 3420,E2 3420} C_VEL
LIN {X 0,Y 704.538,Z 809.06,A -85,B 0,C 180,E1 3424.922,E2 3424.922} C_VEL
LIN {X 0,Y 704.311,Z 809.06,A -85,B 0,C 180,E1 3429.883,E2 3429.883} C_VEL
LIN {X 0,Y 704.199,Z 809.06,A -85,B 0,C 180,E1 3434.45,E2 3434.45} C_VEL
LIN {X 0,Y 700.274,Z 809.06,A -85,B 0,C 180,E1 3435.84,E2 3435.84} C_VEL
LIN {X 0,Y 696.398,Z 809.06,A -85,B 0,C 180,E1 3437.247,E2 3437.247} C_VEL
LIN {X 0,Y 696.244,Z 809.06,A -85,B 0,C 180,E1 3441.65,E2 3441.65} C_VEL
LIN {X 0,Y 696.176,Z 809.06,A -85,B 0,C 180,E1 3445.727,E2 3445.727} C_VEL
LIN {X 0,Y 696.153,Z 809.06,A -85,B 0,C 180,E1 3449.948,E2 3449.948} C_VEL
LIN {X 0,Y 696.128,Z 809.06,A -85,B 0,C 180,E1 3454.418,E2 3454.418} C_VEL
LIN {X 0,Y 696.027,Z 809.06,A -85,B 0,C 180,E1 3459.018,E2 3459.018} C_VEL
LIN {X 0,Y 696.283,Z 809.06,A -85,B 0,C 180,E1 3464.255,E2 3464.255} C_VEL
LIN {X 0,Y 696.151,Z 809.089,A -85,B 0,C 180,E1 3469.087,E2 3469.087} C_VEL
LIN {X 0,Y 698.515,Z 814.688,A -85,B 0,C 180,E1 3469.329,E2 3469.329} C_VEL
LIN {X 0,Y 710.712,Z 836.512,A -85,B 0,C 180,E1 3470.449,E2 3470.449} C_VEL
LIN {X 0,Y 710.083,Z 922.393,A -85,B 0,C 180,E1 3471.612,E2 3471.612} C_VEL
LIN {X 0,Y 708.68,Z 966.529,A -85,B 0,C 180,E1 3472.626,E2 3472.626} C_VEL
LIN {X 0,Y 706.984,Z 1014.295,A -85,B 0,C 180,E1 3474.267,E2 3474.267} C_VEL
LIN {X 0,Y 704.907,Z 1060.91,A -85,B 0,C 180,E1 3476.441,E2 3476.441} C_VEL
LIN {X 0,Y 702.909,Z 1102.566,A -85,B 0,C 180,E1 3478.935,E2 3478.935} C_VEL
LIN {X 0,Y 700.9,Z 1144.772,A -85,B 0,C 180,E1 3482.114,E2 3482.114} C_VEL
LIN {X 0,Y 699.313,Z 1180.156,A -85,B 0,C 180,E1 3485.446,E2 3485.446} C_VEL
LIN {X 0,Y 698.189,Z 1210.558,A -85,B 0,C 180,E1 3488.967,E2 3488.967} C_VEL
LIN {X 0,Y 697.4,Z 1236.265,A -85,B 0,C 180,E1 3492.723,E2 3492.723} C_VEL
LIN {X 0,Y 696.956,Z 1256.529,A -85,B 0,C 180,E1 3496.517,E2 3496.517} C_VEL
LIN {X 0,Y 696.707,Z 1271.809,A -85,B 0,C 180,E1 3500.461,E2 3500.461} C_VEL
LIN {X 0,Y 696.618,Z 1281.789,A -85,B 0,C 180,E1 3504.393,E2 3504.393} C_VEL
LIN {X 0,Y 696.562,Z 1285.871,A -85,B 0,C 180,E1 3507.508,E2 3507.508} C_VEL
LIN {X 0,Y 696.691,Z 1286.67,A -85,B 0,C 180,E1 3511.238,E2 3511.238} C_VEL
LIN {X 0,Y 696.507,Z 1282.919,A -85,B 0,C 180,E1 3514.973,E2 3514.973} C_VEL
LIN {X 0,Y 696.513,Z 1276.117,A -85,B 0,C 180,E1 3518.101,E2 3518.101} C_VEL
LIN {X 0,Y 696.756,Z 1263.413,A -85,B 0,C 180,E1 3521.884,E2 3521.884} C_VEL
LIN {X 0,Y 697.038,Z 1245.474,A -85,B 0,C 180,E1 3525.677,E2 3525.677} C_VEL
LIN {X 0,Y 697.666,Z 1223.113,A -85,B 0,C 180,E1 3529.312,E2 3529.312} C_VEL
LIN {X 0,Y 698.643,Z 1195.213,A -85,B 0,C 180,E1 3532.906,E2 3532.906} C_VEL
LIN {X 0,Y 700.225,Z 1159.916,A -85,B 0,C 180,E1 3536.551,E2 3536.551} C_VEL
LIN {X 0,Y 702.044,Z 1120.586,A -85,B 0,C 180,E1 3539.793,E2 3539.793} C_VEL
LIN {X 0,Y 704.018,Z 1080.697,A -85,B 0,C 180,E1 3542.445,E2 3542.445} C_VEL
LIN {X 0,Y 706.088,Z 1036.757,A -85,B 0,C 180,E1 3544.755,E2 3544.755} C_VEL
LIN {X 0,Y 707.939,Z 992.969,A -85,B 0,C 180,E1 3546.53,E2 3546.53} C_VEL
LIN {X 0,Y 709.305,Z 949.102,A -85,B 0,C 180,E1 3547.828,E2 3547.828} C_VEL
LIN {X 0,Y 710.344,Z 903.652,A -85,B 0,C 180,E1 3548.699,E2 3548.699} C_VEL
LIN {X 0,Y 710.017,Z 835.675,A -85,B 0,C 180,E1 3549.608,E2 3549.608} C_VEL
LIN {X 0,Y 696.209,Z 810.249,A -85,B 0,C 180,E1 3550.894,E2 3550.894} C_VEL
LIN {X 0,Y 696.103,Z 809.06,A -85,B 0,C 180,E1 3550.954,E2 3550.954} C_VEL
LIN {X 0,Y 696.177,Z 809.06,A -85,B 0,C 180,E1 3555.739,E2 3555.739} C_VEL
LIN {X 0,Y 696.119,Z 809.06,A -85,B 0,C 180,E1 3561.385,E2 3561.385} C_VEL
LIN {X 0,Y 696.052,Z 809.06,A -85,B 0,C 180,E1 3565.638,E2 3565.638} C_VEL
LIN {X 0,Y 696.084,Z 809.06,A -85,B 0,C 180,E1 3570.253,E2 3570.253} C_VEL
LIN {X 0,Y 696.133,Z 809.06,A -85,B 0,C 180,E1 3574.271,E2 3574.271} C_VEL
LIN {X 0,Y 696.116,Z 809.06,A -85,B 0,C 180,E1 3579.678,E2 3579.678} C_VEL
LIN {X 0,Y 696.126,Z 809.06,A -85,B 0,C 180,E1 3584.902,E2 3584.902} C_VEL
LIN {X 0,Y 696.169,Z 809.06,A -85,B 0,C 180,E1 3586.559,E2 3586.559} C_VEL
LIN {X 0,Y 707.876,Z 838.736,A -85,B 0,C 180,E1 3588.271,E2 3588.271} C_VEL
LIN {X 0,Y 706.137,Z 885.611,A -85,B 0,C 180,E1 3590.143,E2 3590.143} C_VEL
LIN {X 0,Y 703.859,Z 932.328,A -85,B 0,C 180,E1 3592.599,E2 3592.599} C_VEL
LIN {X 0,Y 701.886,Z 974.362,A -85,B 0,C 180,E1 3595.446,E2 3595.446} C_VEL
LIN {X 0,Y 700.11,Z 1012.097,A -85,B 0,C 180,E1 3598.608,E2 3598.608} C_VEL
LIN {X 0,Y 698.669,Z 1047.61,A -85,B 0,C 180,E1 3602.324,E2 3602.324} C_VEL
LIN {X 0,Y 697.665,Z 1075.814,A -85,B 0,C 180,E1 3606.045,E2 3606.045} C_VEL
LIN {X 0,Y 697.111,Z 1099.291,A -85,B 0,C 180,E1 3609.985,E2 3609.985} C_VEL
LIN {X 0,Y 696.696,Z 1116.216,A -85,B 0,C 180,E1 3613.801,E2 3613.801} C_VEL
LIN {X 0,Y 696.574,Z 1128.22,A -85,B 0,C 180,E1 3617.679,E2 3617.679} C_VEL
LIN {X 0,Y 696.412,Z 1135.18,A -85,B 0,C 180,E1 3621.644,E2 3621.644} C_VEL
LIN {X 0,Y 696.398,Z 1136.814,A -85,B 0,C 180,E1 3625.718,E2 3625.718} C_VEL
LIN {X 0,Y 696.558,Z 1132.906,A -85,B 0,C 180,E1 3629.928,E2 3629.928} C_VEL
LIN {X 0,Y 696.747,Z 1123.39,A -85,B 0,C 180,E1 3633.986,E2 3633.986} C_VEL
LIN {X 0,Y 696.998,Z 1108.453,A -85,B 0,C 180,E1 3638.006,E2 3638.006} C_VEL
LIN {X 0,Y 697.375,Z 1087.808,A -85,B 0,C 180,E1 3641.981,E2 3641.981} C_VEL
LIN {X 0,Y 698.148,Z 1061.384,A -85,B 0,C 180,E1 3645.878,E2 3645.878} C_VEL
LIN {X 0,Y 699.299,Z 1030.395,A -85,B 0,C 180,E1 3649.485,E2 3649.485} C_VEL
LIN {X 0,Y 700.897,Z 994.381,A -85,B 0,C 180,E1 3652.875,E2 3652.875} C_VEL
LIN {X 0,Y 702.939,Z 952.483,A -85,B 0,C 180,E1 3656.026,E2 3656.026} C_VEL
LIN {X 0,Y 705.042,Z 909.705,A -85,B 0,C 180,E1 3658.576,E2 3658.576} C_VEL
LIN {X 0,Y 707,Z 864.514,A -85,B 0,C 180,E1 3660.681,E2 3660.681} C_VEL
LIN {X 0,Y 707.797,Z 836.998,A -85,B 0,C 180,E1 3661.707,E2 3661.707} C_VEL
LIN {X 0,Y 696.168,Z 809.06,A -85,B 0,C 180,E1 3663.411,E2 3663.411} C_VEL
LIN {X 0,Y 696.065,Z 809.06,A -85,B 0,C 180,E1 3668.974,E2 3668.974} C_VEL
LIN {X 0,Y 696.141,Z 809.06,A -85,B 0,C 180,E1 3674.907,E2 3674.907} C_VEL
LIN {X 0,Y 696.459,Z 809.06,A -85,B 0,C 180,E1 3680.01,E2 3680.01} C_VEL
LIN {X 0,Y 696.428,Z 809.06,A -85,B 0,C 180,E1 3685.026,E2 3685.026} C_VEL
LIN {X 0,Y 696.427,Z 809.06,A -85,B 0,C 180,E1 3690.005,E2 3690.005} C_VEL
LIN {X 0,Y 696.557,Z 809.06,A -85,B 0,C 180,E1 3694.983,E2 3694.983} C_VEL
LIN {X 0,Y 696.371,Z 809.06,A -85,B 0,C 180,E1 3700.002,E2 3700.002} C_VEL
LIN {X 0,Y 696.343,Z 809.06,A -85,B 0,C 180,E1 3705.099,E2 3705.099} C_VEL
LIN {X 0,Y 696.342,Z 809.06,A -85,B 0,C 180,E1 3709.001,E2 3709.001} C_VEL
LIN {X 0,Y 696.236,Z 809.06,A -85,B 0,C 180,E1 3714.359,E2 3714.359} C_VEL
LIN {X 0,Y 696.167,Z 809.06,A -85,B 0,C 180,E1 3719.954,E2 3719.954} C_VEL
LIN {X 0,Y 696.159,Z 809.06,A -85,B 0,C 180,E1 3724.435,E2 3724.435} C_VEL
LIN {X 0,Y 696.005,Z 809.06,A -85,B 0,C 180,E1 3729.027,E2 3729.027} C_VEL
LIN {X 0,Y 696.25,Z 809.06,A -85,B 0,C 180,E1 3734.262,E2 3734.262} C_VEL
LIN {X 0,Y 696.062,Z 809.06,A -85,B 0,C 180,E1 3739.454,E2 3739.454} C_VEL
LIN {X 0,Y 696.024,Z 809.06,A -85,B 0,C 180,E1 3744.117,E2 3744.117} C_VEL
LIN {X 0,Y 696.097,Z 809.06,A -85,B 0,C 180,E1 3748.604,E2 3748.604} C_VEL
LIN {X 0,Y 696.312,Z 809.06,A -85,B 0,C 180,E1 3752.891,E2 3752.891} C_VEL
LIN {X 0,Y 696.289,Z 809.06,A -85,B 0,C 180,E1 3758.352,E2 3758.352} C_VEL
LIN {X 0,Y 696.345,Z 809.06,A -85,B 0,C 180,E1 3763.616,E2 3763.616} C_VEL
LIN {X 0,Y 696.399,Z 809.06,A -85,B 0,C 180,E1 3768.74,E2 3768.74} C_VEL
LIN {X 0,Y 696.499,Z 809.06,A -85,B 0,C 180,E1 3773.773,E2 3773.773} C_VEL
LIN {X 0,Y 696.419,Z 809.06,A -85,B 0,C 180,E1 3778.757,E2 3778.757} C_VEL
LIN {X 0,Y 696.452,Z 809.06,A -85,B 0,C 180,E1 3782.487,E2 3782.487} C_VEL
LIN {X 0,Y 696.415,Z 809.06,A -85,B 0,C 180,E1 3786.228,E2 3786.228} C_VEL
LIN {X 0,Y 696.343,Z 809.06,A -85,B 0,C 180,E1 3791.262,E2 3791.262} C_VEL
LIN {X 0,Y 696.392,Z 809.06,A -85,B 0,C 180,E1 3796.384,E2 3796.384} C_VEL
LIN {X 0,Y 696.398,Z 809.06,A -85,B 0,C 180,E1 3797.247,E2 3797.247} C_VEL
LIN {X 0,Y 693.872,Z 809.06,A -85,B 0,C 180,E1 3798.305,E2 3798.305} C_VEL
LIN {X 0,Y 688.428,Z 809.06,A -85,B 0,C 180,E1 3799.886,E2 3799.886} C_VEL
LIN {X 0,Y 688.338,Z 809.06,A -85,B 0,C 180,E1 3800.068,E2 3800.068} C_VEL
LIN {X 0,Y 688.301,Z 809.06,A -85,B 0,C 180,E1 3804.652,E2 3804.652} C_VEL
LIN {X 0,Y 688.247,Z 809.06,A -85,B 0,C 180,E1 3808.881,E2 3808.881} C_VEL
LIN {X 0,Y 688.226,Z 809.06,A -85,B 0,C 180,E1 3813.446,E2 3813.446} C_VEL
LIN {X 0,Y 688.198,Z 809.06,A -85,B 0,C 180,E1 3817.935,E2 3817.935} C_VEL
LIN {X 0,Y 688.332,Z 809.06,A -85,B 0,C 180,E1 3823.572,E2 3823.572} C_VEL
LIN {X 0,Y 688.202,Z 809.06,A -85,B 0,C 180,E1 3828.5,E2 3828.5} C_VEL
LIN {X 0,Y 690.65,Z 814.749,A -85,B 0,C 180,E1 3828.767,E2 3828.767} C_VEL
LIN {X 0,Y 704.688,Z 840.193,A -85,B 0,C 180,E1 3830.091,E2 3830.091} C_VEL
LIN {X 0,Y 703.89,Z 922.276,A -85,B 0,C 180,E1 3831.21,E2 3831.21} C_VEL
LIN {X 0,Y 702.385,Z 965.61,A -85,B 0,C 180,E1 3832.206,E2 3832.206} C_VEL
LIN {X 0,Y 700.564,Z 1012.318,A -85,B 0,C 180,E1 3833.8,E2 3833.8} C_VEL
LIN {X 0,Y 698.279,Z 1058.065,A -85,B 0,C 180,E1 3835.921,E2 3835.921} C_VEL
LIN {X 0,Y 696,Z 1101.107,A -85,B 0,C 180,E1 3838.486,E2 3838.486} C_VEL
LIN {X 0,Y 693.663,Z 1143.046,A -85,B 0,C 180,E1 3841.651,E2 3841.651} C_VEL
LIN {X 0,Y 691.879,Z 1178.339,A -85,B 0,C 180,E1 3844.97,E2 3844.97} C_VEL
LIN {X 0,Y 690.508,Z 1209.996,A -85,B 0,C 180,E1 3848.647,E2 3848.647} C_VEL
LIN {X 0,Y 689.606,Z 1236.175,A -85,B 0,C 180,E1 3852.506,E2 3852.506} C_VEL
LIN {X 0,Y 689.106,Z 1256.526,A -85,B 0,C 180,E1 3856.361,E2 3856.361} C_VEL
LIN {X 0,Y 688.831,Z 1272.036,A -85,B 0,C 180,E1 3860.425,E2 3860.425} C_VEL
LIN {X 0,Y 688.749,Z 1281.789,A -85,B 0,C 180,E1 3864.329,E2 3864.329} C_VEL
LIN {X 0,Y 688.659,Z 1285.871,A -85,B 0,C 180,E1 3867.48,E2 3867.48} C_VEL
LIN {X 0,Y 688.81,Z 1286.67,A -85,B 0,C 180,E1 3871.252,E2 3871.252} C_VEL
LIN {X 0,Y 688.609,Z 1282.919,A -85,B 0,C 180,E1 3875.03,E2 3875.03} C_VEL
LIN {X 0,Y 688.631,Z 1276.117,A -85,B 0,C 180,E1 3878.195,E2 3878.195} C_VEL
LIN {X 0,Y 688.899,Z 1264.694,A -85,B 0,C 180,E1 3881.7,E2 3881.7} C_VEL
LIN {X 0,Y 689.202,Z 1247.195,A -85,B 0,C 180,E1 3885.541,E2 3885.541} C_VEL
LIN {X 0,Y 689.847,Z 1225.521,A -85,B 0,C 180,E1 3889.176,E2 3889.176} C_VEL
LIN {X 0,Y 690.938,Z 1198.12,A -85,B 0,C 180,E1 3892.836,E2 3892.836} C_VEL
LIN {X 0,Y 692.542,Z 1164.304,A -85,B 0,C 180,E1 3896.435,E2 3896.435} C_VEL
LIN {X 0,Y 694.492,Z 1127.776,A -85,B 0,C 180,E1 3899.585,E2 3899.585} C_VEL
LIN {X 0,Y 696.841,Z 1085.454,A -85,B 0,C 180,E1 3902.519,E2 3902.519} C_VEL
LIN {X 0,Y 699.096,Z 1043.097,A -85,B 0,C 180,E1 3904.835,E2 3904.835} C_VEL
LIN {X 0,Y 701.191,Z 998.781,A -85,B 0,C 180,E1 3906.708,E2 3906.708} C_VEL
LIN {X 0,Y 702.892,Z 953.317,A -85,B 0,C 180,E1 3908.123,E2 3908.123} C_VEL
LIN {X 0,Y 704.114,Z 908.611,A -85,B 0,C 180,E1 3909.029,E2 3909.029} C_VEL
LIN {X 0,Y 704.056,Z 839.142,A -85,B 0,C 180,E1 3909.965,E2 3909.965} C_VEL
LIN {X 0,Y 688.295,Z 809.854,A -85,B 0,C 180,E1 3911.472,E2 3911.472} C_VEL
LIN {X 0,Y 688.273,Z 809.06,A -85,B 0,C 180,E1 3915.371,E2 3915.371} C_VEL
LIN {X 0,Y 688.149,Z 809.06,A -85,B 0,C 180,E1 3920.449,E2 3920.449} C_VEL
LIN {X 0,Y 688.129,Z 809.06,A -85,B 0,C 180,E1 3925.186,E2 3925.186} C_VEL
LIN {X 0,Y 688.126,Z 809.06,A -85,B 0,C 180,E1 3929.666,E2 3929.666} C_VEL
LIN {X 0,Y 688.219,Z 809.06,A -85,B 0,C 180,E1 3934.171,E2 3934.171} C_VEL
LIN {X 0,Y 688.2,Z 809.06,A -85,B 0,C 180,E1 3939.433,E2 3939.433} C_VEL
LIN {X 0,Y 688.236,Z 809.06,A -85,B 0,C 180,E1 3945.004,E2 3945.004} C_VEL
LIN {X 0,Y 688.228,Z 809.06,A -85,B 0,C 180,E1 3946.024,E2 3946.024} C_VEL
LIN {X 0,Y 701.35,Z 841.601,A -85,B 0,C 180,E1 3947.973,E2 3947.973} C_VEL
LIN {X 0,Y 699.213,Z 889.953,A -85,B 0,C 180,E1 3949.966,E2 3949.966} C_VEL
LIN {X 0,Y 696.795,Z 934.441,A -85,B 0,C 180,E1 3952.367,E2 3952.367} C_VEL
LIN {X 0,Y 694.62,Z 976.092,A -85,B 0,C 180,E1 3955.242,E2 3955.242} C_VEL
LIN {X 0,Y 692.62,Z 1013.471,A -85,B 0,C 180,E1 3958.437,E2 3958.437} C_VEL
LIN {X 0,Y 691.064,Z 1047.403,A -85,B 0,C 180,E1 3962.036,E2 3962.036} C_VEL
LIN {X 0,Y 689.974,Z 1075.73,A -85,B 0,C 180,E1 3965.813,E2 3965.813} C_VEL
LIN {X 0,Y 689.33,Z 1098.784,A -85,B 0,C 180,E1 3969.713,E2 3969.713} C_VEL
LIN {X 0,Y 688.865,Z 1116.093,A -85,B 0,C 180,E1 3973.638,E2 3973.638} C_VEL
LIN {X 0,Y 688.692,Z 1128.025,A -85,B 0,C 180,E1 3977.513,E2 3977.513} C_VEL
LIN {X 0,Y 688.589,Z 1133.853,A -85,B 0,C 180,E1 3980.554,E2 3980.554} C_VEL
LIN {X 0,Y 688.444,Z 1136.938,A -85,B 0,C 180,E1 3984.645,E2 3984.645} C_VEL
LIN {X 0,Y 688.538,Z 1134.514,A -85,B 0,C 180,E1 3988.867,E2 3988.867} C_VEL
LIN {X 0,Y 688.675,Z 1127.432,A -85,B 0,C 180,E1 3992.644,E2 3992.644} C_VEL
LIN {X 0,Y 688.799,Z 1115.93,A -85,B 0,C 180,E1 3996.319,E2 3996.319} C_VEL
LIN {X 0,Y 689.127,Z 1100.388,A -85,B 0,C 180,E1 3999.883,E2 3999.883} C_VEL
LIN {X 0,Y 689.715,Z 1080.214,A -85,B 0,C 180,E1 4003.427,E2 4003.427} C_VEL
LIN {X 0,Y 690.715,Z 1053.167,A -85,B 0,C 180,E1 4007.169,E2 4007.169} C_VEL
LIN {X 0,Y 692.204,Z 1021.11,A -85,B 0,C 180,E1 4010.731,E2 4010.731} C_VEL
LIN {X 0,Y 694.178,Z 982.939,A -85,B 0,C 180,E1 4014.141,E2 4014.141} C_VEL
LIN {X 0,Y 696.477,Z 941.734,A -85,B 0,C 180,E1 4017.077,E2 4017.077} C_VEL
LIN {X 0,Y 698.823,Z 898.272,A -85,B 0,C 180,E1 4019.542,E2 4019.542} C_VEL
LIN {X 0,Y 700.884,Z 855.437,A -85,B 0,C 180,E1 4021.42,E2 4021.42} C_VEL
LIN {X 0,Y 700.893,Z 839.461,A -85,B 0,C 180,E1 4022.042,E2 4022.042} C_VEL
LIN {X 0,Y 688.251,Z 809.06,A -85,B 0,C 180,E1 4023.916,E2 4023.916} C_VEL
LIN {X 0,Y 688.184,Z 809.06,A -85,B 0,C 180,E1 4029.438,E2 4029.438} C_VEL
LIN {X 0,Y 688.234,Z 809.06,A -85,B 0,C 180,E1 4035.015,E2 4035.015} C_VEL
LIN {X 0,Y 688.54,Z 809.06,A -85,B 0,C 180,E1 4039.894,E2 4039.894} C_VEL
LIN {X 0,Y 688.525,Z 809.06,A -85,B 0,C 180,E1 4044.969,E2 4044.969} C_VEL
LIN {X 0,Y 688.552,Z 809.06,A -85,B 0,C 180,E1 4050.005,E2 4050.005} C_VEL
LIN {X 0,Y 688.641,Z 809.06,A -85,B 0,C 180,E1 4055.04,E2 4055.04} C_VEL
LIN {X 0,Y 688.465,Z 809.06,A -85,B 0,C 180,E1 4060.118,E2 4060.118} C_VEL
LIN {X 0,Y 688.443,Z 809.06,A -85,B 0,C 180,E1 4065.276,E2 4065.276} C_VEL
LIN {X 0,Y 688.395,Z 809.06,A -85,B 0,C 180,E1 4070.566,E2 4070.566} C_VEL
LIN {X 0,Y 688.256,Z 809.06,A -85,B 0,C 180,E1 4076.052,E2 4076.052} C_VEL
LIN {X 0,Y 688.23,Z 809.06,A -85,B 0,C 180,E1 4081.105,E2 4081.105} C_VEL
LIN {X 0,Y 688.198,Z 809.06,A -85,B 0,C 180,E1 4086.364,E2 4086.364} C_VEL
LIN {X 0,Y 688.16,Z 809.06,A -85,B 0,C 180,E1 4091.71,E2 4091.71} C_VEL
LIN {X 0,Y 688.16,Z 809.06,A -85,B 0,C 180,E1 4096.443,E2 4096.443} C_VEL
LIN {X 0,Y 688.153,Z 809.06,A -85,B 0,C 180,E1 4102.239,E2 4102.239} C_VEL
LIN {X 0,Y 688.094,Z 809.06,A -85,B 0,C 180,E1 4106.704,E2 4106.704} C_VEL
LIN {X 0,Y 688.311,Z 809.06,A -85,B 0,C 180,E1 4111.427,E2 4111.427} C_VEL
LIN {X 0,Y 688.352,Z 809.06,A -85,B 0,C 180,E1 4115.351,E2 4115.351} C_VEL
LIN {X 0,Y 688.429,Z 809.06,A -85,B 0,C 180,E1 4120.779,E2 4120.779} C_VEL
LIN {X 0,Y 688.367,Z 809.06,A -85,B 0,C 180,E1 4126.028,E2 4126.028} C_VEL
LIN {X 0,Y 688.468,Z 809.06,A -85,B 0,C 180,E1 4131.163,E2 4131.163} C_VEL
LIN {X 0,Y 688.616,Z 809.06,A -85,B 0,C 180,E1 4136.226,E2 4136.226} C_VEL
LIN {X 0,Y 688.809,Z 809.06,A -85,B 0,C 180,E1 4141.257,E2 4141.257} C_VEL
LIN {X 0,Y 688.507,Z 809.06,A -85,B 0,C 180,E1 4146.3,E2 4146.3} C_VEL
LIN {X 0,Y 688.45,Z 809.06,A -85,B 0,C 180,E1 4151.393,E2 4151.393} C_VEL
LIN {X 0,Y 688.483,Z 809.06,A -85,B 0,C 180,E1 4156.578,E2 4156.578} C_VEL
LIN {X 0,Y 688.338,Z 809.06,A -85,B 0,C 180,E1 4160.068,E2 4160.068} C_VEL
LIN {X 0,Y 687.082,Z 809.06,A -85,B 0,C 180,E1 4160.788,E2 4160.788} C_VEL
LIN {X 0,Y 680.424,Z 809.06,A -85,B 0,C 180,E1 4162.742,E2 4162.742} C_VEL
LIN {X 0,Y 680.331,Z 809.06,A -85,B 0,C 180,E1 4162.927,E2 4162.927} C_VEL
LIN {X 0,Y 680.335,Z 809.06,A -85,B 0,C 180,E1 4167.801,E2 4167.801} C_VEL
LIN {X 0,Y 680.279,Z 809.06,A -85,B 0,C 180,E1 4172.419,E2 4172.419} C_VEL
LIN {X 0,Y 680.264,Z 809.06,A -85,B 0,C 180,E1 4176.894,E2 4176.894} C_VEL
LIN {X 0,Y 680.402,Z 809.06,A -85,B 0,C 180,E1 4182.865,E2 4182.865} C_VEL
LIN {X 0,Y 680.239,Z 809.06,A -85,B 0,C 180,E1 4187.9,E2 4187.9} C_VEL
LIN {X 0,Y 682.847,Z 814.863,A -85,B 0,C 180,E1 4188.192,E2 4188.192} C_VEL
LIN {X 0,Y 698.605,Z 843.387,A -85,B 0,C 180,E1 4189.715,E2 4189.715} C_VEL
LIN {X 0,Y 697.735,Z 922.252,A -85,B 0,C 180,E1 4190.803,E2 4190.803} C_VEL
LIN {X 0,Y 696.061,Z 965.362,A -85,B 0,C 180,E1 4191.794,E2 4191.794} C_VEL
LIN {X 0,Y 694.082,Z 1012.174,A -85,B 0,C 180,E1 4193.401,E2 4193.401} C_VEL
LIN {X 0,Y 691.554,Z 1057.544,A -85,B 0,C 180,E1 4195.514,E2 4195.514} C_VEL
LIN {X 0,Y 689.064,Z 1100.278,A -85,B 0,C 180,E1 4198.071,E2 4198.071} C_VEL
LIN {X 0,Y 686.416,Z 1142.179,A -85,B 0,C 180,E1 4201.249,E2 4201.249} C_VEL
LIN {X 0,Y 684.44,Z 1177.134,A -85,B 0,C 180,E1 4204.548,E2 4204.548} C_VEL
LIN {X 0,Y 682.878,Z 1209.487,A -85,B 0,C 180,E1 4208.331,E2 4208.331} C_VEL
LIN {X 0,Y 681.806,Z 1235.516,A -85,B 0,C 180,E1 4212.188,E2 4212.188} C_VEL
LIN {X 0,Y 681.279,Z 1256.525,A -85,B 0,C 180,E1 4216.201,E2 4216.201} C_VEL
LIN {X 0,Y 680.948,Z 1271.792,A -85,B 0,C 180,E1 4220.232,E2 4220.232} C_VEL
LIN {X 0,Y 680.85,Z 1281.789,A -85,B 0,C 180,E1 4224.263,E2 4224.263} C_VEL
LIN {X 0,Y 680.771,Z 1285.871,A -85,B 0,C 180,E1 4227.45,E2 4227.45} C_VEL
LIN {X 0,Y 680.907,Z 1286.67,A -85,B 0,C 180,E1 4231.266,E2 4231.266} C_VEL
LIN {X 0,Y 680.731,Z 1282.919,A -85,B 0,C 180,E1 4235.089,E2 4235.089} C_VEL
LIN {X 0,Y 680.746,Z 1274.306,A -85,B 0,C 180,E1 4238.933,E2 4238.933} C_VEL
LIN {X 0,Y 681.074,Z 1261.88,A -85,B 0,C 180,E1 4242.535,E2 4242.535} C_VEL
LIN {X 0,Y 681.473,Z 1243.503,A -85,B 0,C 180,E1 4246.416,E2 4246.416} C_VEL
LIN {X 0,Y 682.319,Z 1220.825,A -85,B 0,C 180,E1 4250.109,E2 4250.109} C_VEL
LIN {X 0,Y 683.74,Z 1190.801,A -85,B 0,C 180,E1 4253.953,E2 4253.953} C_VEL
LIN {X 0,Y 685.514,Z 1157.517,A -85,B 0,C 180,E1 4257.39,E2 4257.39} C_VEL
LIN {X 0,Y 687.983,Z 1117.334,A -85,B 0,C 180,E1 4260.724,E2 4260.724} C_VEL
LIN {X 0,Y 690.408,Z 1075.642,A -85,B 0,C 180,E1 4263.479,E2 4263.479} C_VEL
LIN {X 0,Y 693.122,Z 1030.545,A -85,B 0,C 180,E1 4265.816,E2 4265.816} C_VEL
LIN {X 0,Y 695.262,Z 986.766,A -85,B 0,C 180,E1 4267.532,E2 4267.532} C_VEL
LIN {X 0,Y 696.91,Z 944.78,A -85,B 0,C 180,E1 4268.734,E2 4268.734} C_VEL
LIN {X 0,Y 698.154,Z 900.348,A -85,B 0,C 180,E1 4269.555,E2 4269.555} C_VEL
LIN {X 0,Y 698.031,Z 842.37,A -85,B 0,C 180,E1 4270.338,E2 4270.338} C_VEL
LIN {X 0,Y 680.538,Z 810.56,A -85,B 0,C 180,E1 4272.042,E2 4272.042} C_VEL
LIN {X 0,Y 680.369,Z 809.06,A -85,B 0,C 180,E1 4272.155,E2 4272.155} C_VEL
LIN {X 0,Y 680.224,Z 809.06,A -85,B 0,C 180,E1 4277.136,E2 4277.136} C_VEL
LIN {X 0,Y 680.205,Z 809.06,A -85,B 0,C 180,E1 4281.538,E2 4281.538} C_VEL
LIN {X 0,Y 680.167,Z 809.06,A -85,B 0,C 180,E1 4286.263,E2 4286.263} C_VEL
